Fanuc TP program (LS listing): FM204014.ls

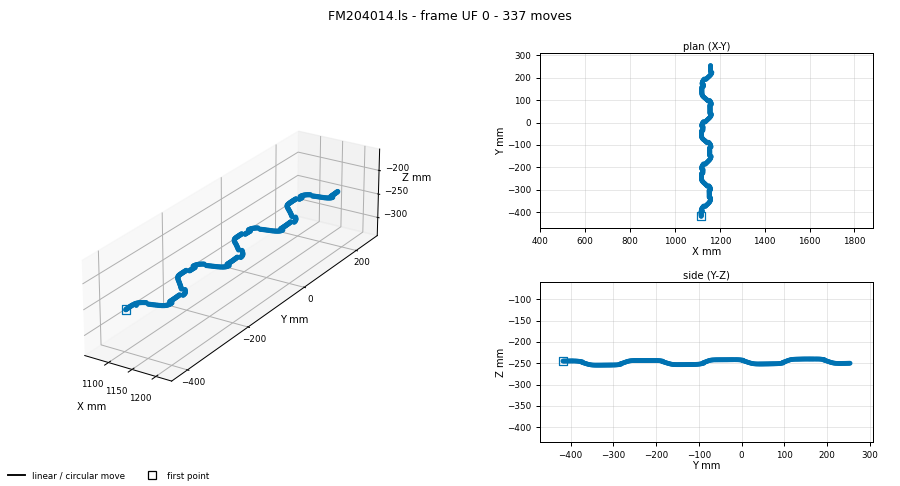
[picture p0: tool path of FM204014.ls in frame UF 0, 337 of 337 moves have a stored position in this frame; points joined in program order, loops and branches not executed]
/PROG  FM204014
/ATTR
OWNER		= MNEDITOR;
COMMENT		= "Auto FANUC move";
PROG_SIZE	= 0;
CREATE		= DATE 26-04-24  TIME 20:40:14;
MODIFIED	= DATE 26-04-24  TIME 20:40:14;
FILE_NAME	= ;
VERSION		= 0;
LINE_COUNT	= 342;
MEMORY_SIZE	= 0;
PROTECT		= READ_WRITE;
TCD:  STACK_SIZE	= 0,
      TASK_PRIORITY	= 50,
      TIME_SLICE	= 0,
      BUSY_LAMP_OFF	= 0,
      ABORT_REQUEST	= 0,
      PAUSE_REQUEST	= 0;
DEFAULT_GROUP	= 1,*,*,*,*;
CONTROL_CODE	= 00000000 00000000;
/MN
   1:  UFRAME_NUM=0 ;
   2:  UTOOL_NUM=1 ;
   3:  R[93]=10 ;
   4:  L P[1] 7mm/sec FINE ;
   5:  L P[2] 7mm/sec CNT50 ;
   6:  L P[3] 7mm/sec CNT50 ;
   7:  L P[4] 7mm/sec CNT50 ;
   8:  L P[5] 7mm/sec CNT50 ;
   9:  L P[6] 7mm/sec CNT50 ;
  10:  L P[7] 7mm/sec CNT50 ;
  11:  L P[8] 7mm/sec CNT50 ;
  12:  L P[9] 7mm/sec CNT50 ;
  13:  L P[10] 7mm/sec CNT50 ;
  14:  L P[11] 7mm/sec CNT50 ;
  15:  L P[12] 7mm/sec CNT50 ;
  16:  L P[13] 7mm/sec CNT50 ;
  17:  L P[14] 7mm/sec CNT50 ;
  18:  L P[15] 7mm/sec CNT50 ;
  19:  L P[16] 7mm/sec CNT50 ;
  20:  L P[17] 7mm/sec CNT50 ;
  21:  L P[18] 7mm/sec CNT50 ;
  22:  L P[19] 7mm/sec CNT50 ;
  23:  L P[20] 7mm/sec CNT50 ;
  24:  L P[21] 7mm/sec CNT50 ;
  25:  L P[22] 7mm/sec CNT50 ;
  26:  L P[23] 7mm/sec CNT50 ;
  27:  L P[24] 7mm/sec CNT50 ;
  28:  L P[25] 7mm/sec CNT50 ;
  29:  L P[26] 7mm/sec CNT50 ;
  30:  L P[27] 7mm/sec CNT50 ;
  31:  L P[28] 7mm/sec CNT50 ;
  32:  L P[29] 7mm/sec CNT50 ;
  33:  L P[30] 7mm/sec CNT50 ;
  34:  L P[31] 7mm/sec CNT50 ;
  35:  L P[32] 7mm/sec CNT50 ;
  36:  L P[33] 7mm/sec CNT50 ;
  37:  L P[34] 7mm/sec CNT50 ;
  38:  L P[35] 7mm/sec CNT50 ;
  39:  L P[36] 7mm/sec CNT50 ;
  40:  L P[37] 7mm/sec CNT50 ;
  41:  L P[38] 7mm/sec CNT50 ;
  42:  L P[39] 7mm/sec CNT50 ;
  43:  L P[40] 7mm/sec CNT50 ;
  44:  L P[41] 7mm/sec CNT50 ;
  45:  L P[42] 7mm/sec CNT50 ;
  46:  L P[43] 7mm/sec CNT50 ;
  47:  L P[44] 7mm/sec CNT50 ;
  48:  L P[45] 7mm/sec CNT50 ;
  49:  L P[46] 7mm/sec CNT50 ;
  50:  L P[47] 7mm/sec CNT50 ;
  51:  L P[48] 7mm/sec CNT50 ;
  52:  L P[49] 7mm/sec CNT50 ;
  53:  L P[50] 7mm/sec CNT50 ;
  54:  L P[51] 7mm/sec CNT50 ;
  55:  L P[52] 7mm/sec CNT50 ;
  56:  L P[53] 7mm/sec CNT50 ;
  57:  L P[54] 7mm/sec CNT50 ;
  58:  L P[55] 7mm/sec CNT50 ;
  59:  L P[56] 7mm/sec CNT50 ;
  60:  L P[57] 7mm/sec CNT50 ;
  61:  L P[58] 7mm/sec CNT50 ;
  62:  L P[59] 7mm/sec CNT50 ;
  63:  L P[60] 7mm/sec CNT50 ;
  64:  L P[61] 7mm/sec CNT50 ;
  65:  L P[62] 7mm/sec CNT50 ;
  66:  L P[63] 7mm/sec CNT50 ;
  67:  L P[64] 7mm/sec CNT50 ;
  68:  L P[65] 7mm/sec CNT50 ;
  69:  L P[66] 7mm/sec CNT50 ;
  70:  L P[67] 7mm/sec CNT50 ;
  71:  L P[68] 7mm/sec CNT50 ;
  72:  L P[69] 7mm/sec CNT50 ;
  73:  L P[70] 7mm/sec CNT50 ;
  74:  L P[71] 7mm/sec CNT50 ;
  75:  L P[72] 7mm/sec CNT50 ;
  76:  L P[73] 7mm/sec CNT50 ;
  77:  L P[74] 7mm/sec CNT50 ;
  78:  L P[75] 7mm/sec CNT50 ;
  79:  L P[76] 7mm/sec CNT50 ;
  80:  L P[77] 7mm/sec CNT50 ;
  81:  L P[78] 7mm/sec CNT50 ;
  82:  L P[79] 7mm/sec CNT50 ;
  83:  L P[80] 7mm/sec CNT50 ;
  84:  L P[81] 7mm/sec CNT50 ;
  85:  L P[82] 7mm/sec CNT50 ;
  86:  L P[83] 7mm/sec CNT50 ;
  87:  L P[84] 7mm/sec CNT50 ;
  88:  L P[85] 7mm/sec CNT50 ;
  89:  L P[86] 7mm/sec CNT50 ;
  90:  L P[87] 7mm/sec CNT50 ;
  91:  L P[88] 7mm/sec CNT50 ;
  92:  L P[89] 7mm/sec CNT50 ;
  93:  L P[90] 7mm/sec CNT50 ;
  94:  L P[91] 7mm/sec CNT50 ;
  95:  L P[92] 7mm/sec CNT50 ;
  96:  L P[93] 7mm/sec CNT50 ;
  97:  L P[94] 7mm/sec CNT50 ;
  98:  L P[95] 7mm/sec CNT50 ;
  99:  L P[96] 7mm/sec CNT50 ;
 100:  L P[97] 7mm/sec CNT50 ;
 101:  L P[98] 7mm/sec CNT50 ;
 102:  L P[99] 7mm/sec CNT50 ;
 103:  L P[100] 7mm/sec CNT50 ;
 104:  L P[101] 7mm/sec CNT50 ;
 105:  L P[102] 7mm/sec CNT50 ;
 106:  L P[103] 7mm/sec CNT50 ;
 107:  L P[104] 7mm/sec CNT50 ;
 108:  L P[105] 7mm/sec CNT50 ;
 109:  L P[106] 7mm/sec CNT50 ;
 110:  L P[107] 7mm/sec CNT50 ;
 111:  L P[108] 7mm/sec CNT50 ;
 112:  L P[109] 7mm/sec CNT50 ;
 113:  L P[110] 7mm/sec CNT50 ;
 114:  L P[111] 7mm/sec CNT50 ;
 115:  L P[112] 7mm/sec CNT50 ;
 116:  L P[113] 7mm/sec CNT50 ;
 117:  L P[114] 7mm/sec CNT50 ;
 118:  L P[115] 7mm/sec CNT50 ;
 119:  L P[116] 7mm/sec CNT50 ;
 120:  L P[117] 7mm/sec CNT50 ;
 121:  L P[118] 7mm/sec CNT50 ;
 122:  L P[119] 7mm/sec CNT50 ;
 123:  L P[120] 7mm/sec CNT50 ;
 124:  L P[121] 7mm/sec CNT50 ;
 125:  L P[122] 7mm/sec CNT50 ;
 126:  L P[123] 7mm/sec CNT50 ;
 127:  L P[124] 7mm/sec CNT50 ;
 128:  L P[125] 7mm/sec CNT50 ;
 129:  L P[126] 7mm/sec CNT50 ;
 130:  L P[127] 7mm/sec CNT50 ;
 131:  L P[128] 7mm/sec CNT50 ;
 132:  L P[129] 7mm/sec CNT50 ;
 133:  L P[130] 7mm/sec CNT50 ;
 134:  L P[131] 7mm/sec CNT50 ;
 135:  L P[132] 7mm/sec CNT50 ;
 136:  L P[133] 7mm/sec CNT50 ;
 137:  L P[134] 7mm/sec CNT50 ;
 138:  L P[135] 7mm/sec CNT50 ;
 139:  L P[136] 7mm/sec CNT50 ;
 140:  L P[137] 7mm/sec CNT50 ;
 141:  L P[138] 7mm/sec CNT50 ;
 142:  L P[139] 7mm/sec CNT50 ;
 143:  L P[140] 7mm/sec CNT50 ;
 144:  L P[141] 7mm/sec CNT50 ;
 145:  L P[142] 7mm/sec CNT50 ;
 146:  L P[143] 7mm/sec CNT50 ;
 147:  L P[144] 7mm/sec CNT50 ;
 148:  L P[145] 7mm/sec CNT50 ;
 149:  L P[146] 7mm/sec CNT50 ;
 150:  L P[147] 7mm/sec CNT50 ;
 151:  L P[148] 7mm/sec CNT50 ;
 152:  L P[149] 7mm/sec CNT50 ;
 153:  L P[150] 7mm/sec CNT50 ;
 154:  L P[151] 7mm/sec CNT50 ;
 155:  L P[152] 7mm/sec CNT50 ;
 156:  L P[153] 7mm/sec CNT50 ;
 157:  L P[154] 7mm/sec CNT50 ;
 158:  L P[155] 7mm/sec CNT50 ;
 159:  L P[156] 7mm/sec CNT50 ;
 160:  L P[157] 7mm/sec CNT50 ;
 161:  L P[158] 7mm/sec CNT50 ;
 162:  L P[159] 7mm/sec CNT50 ;
 163:  L P[160] 7mm/sec CNT50 ;
 164:  L P[161] 7mm/sec CNT50 ;
 165:  L P[162] 7mm/sec CNT50 ;
 166:  L P[163] 7mm/sec CNT50 ;
 167:  L P[164] 7mm/sec CNT50 ;
 168:  L P[165] 7mm/sec CNT50 ;
 169:  L P[166] 7mm/sec CNT50 ;
 170:  L P[167] 7mm/sec CNT50 ;
 171:  L P[168] 7mm/sec CNT50 ;
 172:  L P[169] 7mm/sec CNT50 ;
 173:  L P[170] 7mm/sec CNT50 ;
 174:  L P[171] 7mm/sec CNT50 ;
 175:  L P[172] 7mm/sec CNT50 ;
 176:  L P[173] 7mm/sec CNT50 ;
 177:  L P[174] 7mm/sec CNT50 ;
 178:  L P[175] 7mm/sec CNT50 ;
 179:  L P[176] 7mm/sec CNT50 ;
 180:  L P[177] 7mm/sec CNT50 ;
 181:  L P[178] 7mm/sec CNT50 ;
 182:  L P[179] 7mm/sec CNT50 ;
 183:  L P[180] 7mm/sec CNT50 ;
 184:  L P[181] 7mm/sec CNT50 ;
 185:  L P[182] 7mm/sec CNT50 ;
 186:  L P[183] 7mm/sec CNT50 ;
 187:  L P[184] 7mm/sec CNT50 ;
 188:  L P[185] 7mm/sec CNT50 ;
 189:  L P[186] 7mm/sec CNT50 ;
 190:  L P[187] 7mm/sec CNT50 ;
 191:  L P[188] 7mm/sec CNT50 ;
 192:  L P[189] 7mm/sec CNT50 ;
 193:  L P[190] 7mm/sec CNT50 ;
 194:  L P[191] 7mm/sec CNT50 ;
 195:  L P[192] 7mm/sec CNT50 ;
 196:  L P[193] 7mm/sec CNT50 ;
 197:  L P[194] 7mm/sec CNT50 ;
 198:  L P[195] 7mm/sec CNT50 ;
 199:  L P[196] 7mm/sec CNT50 ;
 200:  L P[197] 7mm/sec CNT50 ;
 201:  L P[198] 7mm/sec CNT50 ;
 202:  L P[199] 7mm/sec CNT50 ;
 203:  L P[200] 7mm/sec CNT50 ;
 204:  L P[201] 7mm/sec CNT50 ;
 205:  L P[202] 7mm/sec CNT50 ;
 206:  L P[203] 7mm/sec CNT50 ;
 207:  L P[204] 7mm/sec CNT50 ;
 208:  L P[205] 7mm/sec CNT50 ;
 209:  L P[206] 7mm/sec CNT50 ;
 210:  L P[207] 7mm/sec CNT50 ;
 211:  L P[208] 7mm/sec CNT50 ;
 212:  L P[209] 7mm/sec CNT50 ;
 213:  L P[210] 7mm/sec CNT50 ;
 214:  L P[211] 7mm/sec CNT50 ;
 215:  L P[212] 7mm/sec CNT50 ;
 216:  L P[213] 7mm/sec CNT50 ;
 217:  L P[214] 7mm/sec CNT50 ;
 218:  L P[215] 7mm/sec CNT50 ;
 219:  L P[216] 7mm/sec CNT50 ;
 220:  L P[217] 7mm/sec CNT50 ;
 221:  L P[218] 7mm/sec CNT50 ;
 222:  L P[219] 7mm/sec CNT50 ;
 223:  L P[220] 7mm/sec CNT50 ;
 224:  L P[221] 7mm/sec CNT50 ;
 225:  L P[222] 7mm/sec CNT50 ;
 226:  L P[223] 7mm/sec CNT50 ;
 227:  L P[224] 7mm/sec CNT50 ;
 228:  L P[225] 7mm/sec CNT50 ;
 229:  L P[226] 7mm/sec CNT50 ;
 230:  L P[227] 7mm/sec CNT50 ;
 231:  L P[228] 7mm/sec CNT50 ;
 232:  L P[229] 7mm/sec CNT50 ;
 233:  L P[230] 7mm/sec CNT50 ;
 234:  L P[231] 7mm/sec CNT50 ;
 235:  L P[232] 7mm/sec CNT50 ;
 236:  L P[233] 7mm/sec CNT50 ;
 237:  L P[234] 7mm/sec CNT50 ;
 238:  L P[235] 7mm/sec CNT50 ;
 239:  L P[236] 7mm/sec CNT50 ;
 240:  L P[237] 7mm/sec CNT50 ;
 241:  L P[238] 7mm/sec CNT50 ;
 242:  L P[239] 7mm/sec CNT50 ;
 243:  L P[240] 7mm/sec CNT50 ;
 244:  L P[241] 7mm/sec CNT50 ;
 245:  L P[242] 7mm/sec CNT50 ;
 246:  L P[243] 7mm/sec CNT50 ;
 247:  L P[244] 7mm/sec CNT50 ;
 248:  L P[245] 7mm/sec CNT50 ;
 249:  L P[246] 7mm/sec CNT50 ;
 250:  L P[247] 7mm/sec CNT50 ;
 251:  L P[248] 7mm/sec CNT50 ;
 252:  L P[249] 7mm/sec CNT50 ;
 253:  L P[250] 7mm/sec CNT50 ;
 254:  L P[251] 7mm/sec CNT50 ;
 255:  L P[252] 7mm/sec CNT50 ;
 256:  L P[253] 7mm/sec CNT50 ;
 257:  L P[254] 7mm/sec CNT50 ;
 258:  L P[255] 7mm/sec CNT50 ;
 259:  L P[256] 7mm/sec CNT50 ;
 260:  L P[257] 7mm/sec CNT50 ;
 261:  L P[258] 7mm/sec CNT50 ;
 262:  L P[259] 7mm/sec CNT50 ;
 263:  L P[260] 7mm/sec CNT50 ;
 264:  L P[261] 7mm/sec CNT50 ;
 265:  L P[262] 7mm/sec CNT50 ;
 266:  L P[263] 7mm/sec CNT50 ;
 267:  L P[264] 7mm/sec CNT50 ;
 268:  L P[265] 7mm/sec CNT50 ;
 269:  L P[266] 7mm/sec CNT50 ;
 270:  L P[267] 7mm/sec CNT50 ;
 271:  L P[268] 7mm/sec CNT50 ;
 272:  L P[269] 7mm/sec CNT50 ;
 273:  L P[270] 7mm/sec CNT50 ;
 274:  L P[271] 7mm/sec CNT50 ;
 275:  L P[272] 7mm/sec CNT50 ;
 276:  L P[273] 7mm/sec CNT50 ;
 277:  L P[274] 7mm/sec CNT50 ;
 278:  L P[275] 7mm/sec CNT50 ;
 279:  L P[276] 7mm/sec CNT50 ;
 280:  L P[277] 7mm/sec CNT50 ;
 281:  L P[278] 7mm/sec CNT50 ;
 282:  L P[279] 7mm/sec CNT50 ;
 283:  L P[280] 7mm/sec CNT50 ;
 284:  L P[281] 7mm/sec CNT50 ;
 285:  L P[282] 7mm/sec CNT50 ;
 286:  L P[283] 7mm/sec CNT50 ;
 287:  L P[284] 7mm/sec CNT50 ;
 288:  L P[285] 7mm/sec CNT50 ;
 289:  L P[286] 7mm/sec CNT50 ;
 290:  L P[287] 7mm/sec CNT50 ;
 291:  L P[288] 7mm/sec CNT50 ;
 292:  L P[289] 7mm/sec CNT50 ;
 293:  L P[290] 7mm/sec CNT50 ;
 294:  L P[291] 7mm/sec CNT50 ;
 295:  L P[292] 7mm/sec CNT50 ;
 296:  L P[293] 7mm/sec CNT50 ;
 297:  L P[294] 7mm/sec CNT50 ;
 298:  L P[295] 7mm/sec CNT50 ;
 299:  L P[296] 7mm/sec CNT50 ;
 300:  L P[297] 7mm/sec CNT50 ;
 301:  L P[298] 7mm/sec CNT50 ;
 302:  L P[299] 7mm/sec CNT50 ;
 303:  L P[300] 7mm/sec CNT50 ;
 304:  L P[301] 7mm/sec CNT50 ;
 305:  L P[302] 7mm/sec CNT50 ;
 306:  L P[303] 7mm/sec CNT50 ;
 307:  L P[304] 7mm/sec CNT50 ;
 308:  L P[305] 7mm/sec CNT50 ;
 309:  L P[306] 7mm/sec CNT50 ;
 310:  L P[307] 7mm/sec CNT50 ;
 311:  L P[308] 7mm/sec CNT50 ;
 312:  L P[309] 7mm/sec CNT50 ;
 313:  L P[310] 7mm/sec CNT50 ;
 314:  L P[311] 7mm/sec CNT50 ;
 315:  L P[312] 7mm/sec CNT50 ;
 316:  L P[313] 7mm/sec CNT50 ;
 317:  L P[314] 7mm/sec CNT50 ;
 318:  L P[315] 7mm/sec CNT50 ;
 319:  L P[316] 7mm/sec CNT50 ;
 320:  L P[317] 7mm/sec CNT50 ;
 321:  L P[318] 7mm/sec CNT50 ;
 322:  L P[319] 7mm/sec CNT50 ;
 323:  L P[320] 7mm/sec CNT50 ;
 324:  L P[321] 7mm/sec CNT50 ;
 325:  L P[322] 7mm/sec CNT50 ;
 326:  L P[323] 7mm/sec CNT50 ;
 327:  L P[324] 7mm/sec CNT50 ;
 328:  L P[325] 7mm/sec CNT50 ;
 329:  L P[326] 7mm/sec CNT50 ;
 330:  L P[327] 7mm/sec CNT50 ;
 331:  L P[328] 7mm/sec CNT50 ;
 332:  L P[329] 7mm/sec CNT50 ;
 333:  L P[330] 7mm/sec CNT50 ;
 334:  L P[331] 7mm/sec CNT50 ;
 335:  L P[332] 7mm/sec CNT50 ;
 336:  L P[333] 7mm/sec CNT50 ;
 337:  L P[334] 7mm/sec CNT50 ;
 338:  L P[335] 7mm/sec CNT50 ;
 339:  L P[336] 7mm/sec CNT50 ;
 340:  L P[337] 7mm/sec FINE ;
 341:  R[93]=1 ;
 342:  END ;
/POS
P[1]{
   GP1:
	UF : 0, UT : 1,		CONFIG : 'N U T, 0, 0, 0',
	X = 1117.340  mm,	Y = -418.120  mm,	Z = -244.843  mm,
	W = 0.000 deg,	P = 30.000 deg,	R = 175.540 deg
};
P[2]{
   GP1:
	UF : 0, UT : 1,		CONFIG : 'N U T, 0, 0, 0',
	X = 1117.260  mm,	Y = -416.121  mm,	Z = -244.824  mm,
	W = 0.000 deg,	P = 30.000 deg,	R = 175.540 deg
};
P[3]{
   GP1:
	UF : 0, UT : 1,		CONFIG : 'N U T, 0, 0, 0',
	X = 1117.178  mm,	Y = -414.124  mm,	Z = -244.789  mm,
	W = 0.000 deg,	P = 30.000 deg,	R = 175.540 deg
};
P[4]{
   GP1:
	UF : 0, UT : 1,		CONFIG : 'N U T, 0, 0, 0',
	X = 1117.094  mm,	Y = -412.119  mm,	Z = -244.747  mm,
	W = 0.000 deg,	P = 30.000 deg,	R = 175.540 deg
};
P[5]{
   GP1:
	UF : 0, UT : 1,		CONFIG : 'N U T, 0, 0, 0',
	X = 1117.019  mm,	Y = -410.103  mm,	Z = -244.710  mm,
	W = 0.000 deg,	P = 30.000 deg,	R = 175.540 deg
};
P[6]{
   GP1:
	UF : 0, UT : 1,		CONFIG : 'N U T, 0, 0, 0',
	X = 1116.955  mm,	Y = -408.082  mm,	Z = -244.672  mm,
	W = 0.000 deg,	P = 30.000 deg,	R = 175.540 deg
};
P[7]{
   GP1:
	UF : 0, UT : 1,		CONFIG : 'N U T, 0, 0, 0',
	X = 1116.909  mm,	Y = -406.055  mm,	Z = -244.633  mm,
	W = 0.000 deg,	P = 30.000 deg,	R = 175.540 deg
};
P[8]{
   GP1:
	UF : 0, UT : 1,		CONFIG : 'N U T, 0, 0, 0',
	X = 1116.881  mm,	Y = -404.021  mm,	Z = -244.596  mm,
	W = 0.000 deg,	P = 30.000 deg,	R = 175.540 deg
};
P[9]{
   GP1:
	UF : 0, UT : 1,		CONFIG : 'N U T, 0, 0, 0',
	X = 1116.880  mm,	Y = -401.987  mm,	Z = -244.564  mm,
	W = 0.000 deg,	P = 30.000 deg,	R = 175.540 deg
};
P[10]{
   GP1:
	UF : 0, UT : 1,		CONFIG : 'N U T, 0, 0, 0',
	X = 1116.899  mm,	Y = -399.955  mm,	Z = -244.547  mm,
	W = 0.000 deg,	P = 30.000 deg,	R = 175.540 deg
};
P[11]{
   GP1:
	UF : 0, UT : 1,		CONFIG : 'N U T, 0, 0, 0',
	X = 1116.941  mm,	Y = -397.902  mm,	Z = -244.542  mm,
	W = 0.000 deg,	P = 30.000 deg,	R = 175.540 deg
};
P[12]{
   GP1:
	UF : 0, UT : 1,		CONFIG : 'N U T, 0, 0, 0',
	X = 1117.034  mm,	Y = -395.846  mm,	Z = -244.547  mm,
	W = 0.000 deg,	P = 30.000 deg,	R = 175.540 deg
};
P[13]{
   GP1:
	UF : 0, UT : 1,		CONFIG : 'N U T, 0, 0, 0',
	X = 1123.135  mm,	Y = -394.244  mm,	Z = -244.557  mm,
	W = 0.000 deg,	P = 30.000 deg,	R = 175.540 deg
};
P[14]{
   GP1:
	UF : 0, UT : 1,		CONFIG : 'N U T, 0, 0, 0',
	X = 1117.391  mm,	Y = -391.546  mm,	Z = -244.600  mm,
	W = 0.000 deg,	P = 30.000 deg,	R = 169.940 deg
};
P[15]{
   GP1:
	UF : 0, UT : 1,		CONFIG : 'N U T, 0, 0, 0',
	X = 1117.843  mm,	Y = -389.291  mm,	Z = -244.691  mm,
	W = 0.000 deg,	P = 30.000 deg,	R = 162.053 deg
};
P[16]{
   GP1:
	UF : 0, UT : 1,		CONFIG : 'N U T, 0, 0, 0',
	X = 1118.496  mm,	Y = -387.015  mm,	Z = -244.808  mm,
	W = 0.000 deg,	P = 30.000 deg,	R = 154.006 deg
};
P[17]{
   GP1:
	UF : 0, UT : 1,		CONFIG : 'N U T, 0, 0, 0',
	X = 1119.426  mm,	Y = -384.740  mm,	Z = -244.961  mm,
	W = 0.000 deg,	P = 30.000 deg,	R = 145.637 deg
};
P[18]{
   GP1:
	UF : 0, UT : 1,		CONFIG : 'N U T, 0, 0, 0',
	X = 1120.551  mm,	Y = -382.554  mm,	Z = -245.152  mm,
	W = 0.000 deg,	P = 30.000 deg,	R = 136.915 deg
};
P[19]{
   GP1:
	UF : 0, UT : 1,		CONFIG : 'N U T, 0, 0, 0',
	X = 1121.835  mm,	Y = -380.363  mm,	Z = -245.385  mm,
	W = 0.000 deg,	P = 30.000 deg,	R = 136.915 deg
};
P[20]{
   GP1:
	UF : 0, UT : 1,		CONFIG : 'N U T, 0, 0, 0',
	X = 1123.398  mm,	Y = -378.182  mm,	Z = -245.708  mm,
	W = 0.000 deg,	P = 30.000 deg,	R = 136.915 deg
};
P[21]{
   GP1:
	UF : 0, UT : 1,		CONFIG : 'N U T, 0, 0, 0',
	X = 1125.083  mm,	Y = -376.092  mm,	Z = -246.105  mm,
	W = 0.000 deg,	P = 30.000 deg,	R = 136.915 deg
};
P[22]{
   GP1:
	UF : 0, UT : 1,		CONFIG : 'N U T, 0, 0, 0',
	X = 1126.825  mm,	Y = -374.022  mm,	Z = -246.540  mm,
	W = 0.000 deg,	P = 30.000 deg,	R = 136.915 deg
};
P[23]{
   GP1:
	UF : 0, UT : 1,		CONFIG : 'N U T, 0, 0, 0',
	X = 1128.702  mm,	Y = -371.963  mm,	Z = -247.047  mm,
	W = 0.000 deg,	P = 30.000 deg,	R = 136.915 deg
};
P[24]{
   GP1:
	UF : 0, UT : 1,		CONFIG : 'N U T, 0, 0, 0',
	X = 1134.942  mm,	Y = -374.080  mm,	Z = -247.615  mm,
	W = 0.000 deg,	P = 30.000 deg,	R = 136.915 deg
};
P[25]{
   GP1:
	UF : 0, UT : 1,		CONFIG : 'N U T, 0, 0, 0',
	X = 1136.860  mm,	Y = -372.134  mm,	Z = -248.238  mm,
	W = 0.000 deg,	P = 30.000 deg,	R = 136.915 deg
};
P[26]{
   GP1:
	UF : 0, UT : 1,		CONFIG : 'N U T, 0, 0, 0',
	X = 1138.910  mm,	Y = -370.162  mm,	Z = -248.902  mm,
	W = 0.000 deg,	P = 30.000 deg,	R = 136.915 deg
};
P[27]{
   GP1:
	UF : 0, UT : 1,		CONFIG : 'N U T, 0, 0, 0',
	X = 1140.982  mm,	Y = -368.168  mm,	Z = -249.556  mm,
	W = 0.000 deg,	P = 30.000 deg,	R = 136.915 deg
};
P[28]{
   GP1:
	UF : 0, UT : 1,		CONFIG : 'N U T, 0, 0, 0',
	X = 1143.070  mm,	Y = -366.183  mm,	Z = -250.199  mm,
	W = 0.000 deg,	P = 30.000 deg,	R = 136.915 deg
};
P[29]{
   GP1:
	UF : 0, UT : 1,		CONFIG : 'N U T, 0, 0, 0',
	X = 1145.207  mm,	Y = -364.186  mm,	Z = -250.847  mm,
	W = 0.000 deg,	P = 30.000 deg,	R = 136.915 deg
};
P[30]{
   GP1:
	UF : 0, UT : 1,		CONFIG : 'N U T, 0, 0, 0',
	X = 1147.334  mm,	Y = -362.176  mm,	Z = -251.475  mm,
	W = 0.000 deg,	P = 30.000 deg,	R = 143.608 deg
};
P[31]{
   GP1:
	UF : 0, UT : 1,		CONFIG : 'N U T, 0, 0, 0',
	X = 1149.502  mm,	Y = -360.107  mm,	Z = -252.087  mm,
	W = 0.000 deg,	P = 30.000 deg,	R = 156.114 deg
};
P[32]{
   GP1:
	UF : 0, UT : 1,		CONFIG : 'N U T, 0, 0, 0',
	X = 1151.458  mm,	Y = -357.994  mm,	Z = -252.623  mm,
	W = 0.000 deg,	P = 30.000 deg,	R = 167.837 deg
};
P[33]{
   GP1:
	UF : 0, UT : 1,		CONFIG : 'N U T, 0, 0, 0',
	X = 1153.272  mm,	Y = -355.871  mm,	Z = -253.109  mm,
	W = 0.000 deg,	P = 30.000 deg,	R = 179.135 deg
};
P[34]{
   GP1:
	UF : 0, UT : 1,		CONFIG : 'N U T, 0, 0, 0',
	X = 1154.901  mm,	Y = -353.669  mm,	Z = -253.519  mm,
	W = 0.000 deg,	P = 30.000 deg,	R = 179.135 deg
};
P[35]{
   GP1:
	UF : 0, UT : 1,		CONFIG : 'N U T, 0, 0, 0',
	X = 1156.258  mm,	Y = -351.400  mm,	Z = -253.841  mm,
	W = 0.000 deg,	P = 30.000 deg,	R = 179.135 deg
};
P[36]{
   GP1:
	UF : 0, UT : 1,		CONFIG : 'N U T, 0, 0, 0',
	X = 1157.318  mm,	Y = -349.081  mm,	Z = -254.072  mm,
	W = 0.000 deg,	P = 30.000 deg,	R = 179.135 deg
};
P[37]{
   GP1:
	UF : 0, UT : 1,		CONFIG : 'N U T, 0, 0, 0',
	X = 1158.065  mm,	Y = -346.706  mm,	Z = -254.224  mm,
	W = 0.000 deg,	P = 30.000 deg,	R = 179.135 deg
};
P[38]{
   GP1:
	UF : 0, UT : 1,		CONFIG : 'N U T, 0, 0, 0',
	X = 1158.455  mm,	Y = -344.449  mm,	Z = -254.296  mm,
	W = 0.000 deg,	P = 30.000 deg,	R = 179.135 deg
};
P[39]{
   GP1:
	UF : 0, UT : 1,		CONFIG : 'N U T, 0, 0, 0',
	X = 1158.742  mm,	Y = -342.283  mm,	Z = -254.346  mm,
	W = 0.000 deg,	P = 30.000 deg,	R = 179.135 deg
};
P[40]{
   GP1:
	UF : 0, UT : 1,		CONFIG : 'N U T, 0, 0, 0',
	X = 1158.865  mm,	Y = -340.124  mm,	Z = -254.355  mm,
	W = 0.000 deg,	P = 30.000 deg,	R = 179.135 deg
};
P[41]{
   GP1:
	UF : 0, UT : 1,		CONFIG : 'N U T, 0, 0, 0',
	X = 1158.920  mm,	Y = -338.068  mm,	Z = -254.355  mm,
	W = 0.000 deg,	P = 30.000 deg,	R = 179.135 deg
};
P[42]{
   GP1:
	UF : 0, UT : 1,		CONFIG : 'N U T, 0, 0, 0',
	X = 1158.958  mm,	Y = -336.046  mm,	Z = -254.353  mm,
	W = 0.000 deg,	P = 30.000 deg,	R = 179.135 deg
};
P[43]{
   GP1:
	UF : 0, UT : 1,		CONFIG : 'N U T, 0, 0, 0',
	X = 1152.982  mm,	Y = -333.969  mm,	Z = -254.350  mm,
	W = 0.000 deg,	P = 30.000 deg,	R = 179.135 deg
};
P[44]{
   GP1:
	UF : 0, UT : 1,		CONFIG : 'N U T, 0, 0, 0',
	X = 1153.000  mm,	Y = -331.976  mm,	Z = -254.343  mm,
	W = 0.000 deg,	P = 30.000 deg,	R = 179.135 deg
};
P[45]{
   GP1:
	UF : 0, UT : 1,		CONFIG : 'N U T, 0, 0, 0',
	X = 1153.014  mm,	Y = -329.984  mm,	Z = -254.328  mm,
	W = 0.000 deg,	P = 30.000 deg,	R = 179.135 deg
};
P[46]{
   GP1:
	UF : 0, UT : 1,		CONFIG : 'N U T, 0, 0, 0',
	X = 1153.021  mm,	Y = -327.991  mm,	Z = -254.312  mm,
	W = 0.000 deg,	P = 30.000 deg,	R = 179.135 deg
};
P[47]{
   GP1:
	UF : 0, UT : 1,		CONFIG : 'N U T, 0, 0, 0',
	X = 1153.026  mm,	Y = -325.995  mm,	Z = -254.292  mm,
	W = 0.000 deg,	P = 30.000 deg,	R = 179.135 deg
};
P[48]{
   GP1:
	UF : 0, UT : 1,		CONFIG : 'N U T, 0, 0, 0',
	X = 1153.029  mm,	Y = -323.998  mm,	Z = -254.272  mm,
	W = 0.000 deg,	P = 30.000 deg,	R = 179.135 deg
};
P[49]{
   GP1:
	UF : 0, UT : 1,		CONFIG : 'N U T, 0, 0, 0',
	X = 1153.029  mm,	Y = -322.001  mm,	Z = -254.251  mm,
	W = 0.000 deg,	P = 30.000 deg,	R = 179.135 deg
};
P[50]{
   GP1:
	UF : 0, UT : 1,		CONFIG : 'N U T, 0, 0, 0',
	X = 1153.027  mm,	Y = -320.008  mm,	Z = -254.230  mm,
	W = 0.000 deg,	P = 30.000 deg,	R = 179.135 deg
};
P[51]{
   GP1:
	UF : 0, UT : 1,		CONFIG : 'N U T, 0, 0, 0',
	X = 1153.018  mm,	Y = -318.016  mm,	Z = -254.210  mm,
	W = 0.000 deg,	P = 30.000 deg,	R = 179.135 deg
};
P[52]{
   GP1:
	UF : 0, UT : 1,		CONFIG : 'N U T, 0, 0, 0',
	X = 1153.005  mm,	Y = -316.026  mm,	Z = -254.197  mm,
	W = 0.000 deg,	P = 30.000 deg,	R = 179.135 deg
};
P[53]{
   GP1:
	UF : 0, UT : 1,		CONFIG : 'N U T, 0, 0, 0',
	X = 1152.983  mm,	Y = -314.037  mm,	Z = -254.183  mm,
	W = 0.000 deg,	P = 30.000 deg,	R = 179.135 deg
};
P[54]{
   GP1:
	UF : 0, UT : 1,		CONFIG : 'N U T, 0, 0, 0',
	X = 1152.956  mm,	Y = -312.053  mm,	Z = -254.171  mm,
	W = 0.000 deg,	P = 30.000 deg,	R = 179.135 deg
};
P[55]{
   GP1:
	UF : 0, UT : 1,		CONFIG : 'N U T, 0, 0, 0',
	X = 1152.913  mm,	Y = -310.069  mm,	Z = -254.154  mm,
	W = 0.000 deg,	P = 30.000 deg,	R = 179.135 deg
};
P[56]{
   GP1:
	UF : 0, UT : 1,		CONFIG : 'N U T, 0, 0, 0',
	X = 1152.865  mm,	Y = -308.079  mm,	Z = -254.132  mm,
	W = 0.000 deg,	P = 30.000 deg,	R = 179.135 deg
};
P[57]{
   GP1:
	UF : 0, UT : 1,		CONFIG : 'N U T, 0, 0, 0',
	X = 1152.808  mm,	Y = -306.093  mm,	Z = -254.108  mm,
	W = 0.000 deg,	P = 30.000 deg,	R = 179.135 deg
};
P[58]{
   GP1:
	UF : 0, UT : 1,		CONFIG : 'N U T, 0, 0, 0',
	X = 1152.742  mm,	Y = -304.113  mm,	Z = -254.081  mm,
	W = 0.000 deg,	P = 30.000 deg,	R = 179.135 deg
};
P[59]{
   GP1:
	UF : 0, UT : 1,		CONFIG : 'N U T, 0, 0, 0',
	X = 1152.659  mm,	Y = -302.131  mm,	Z = -254.050  mm,
	W = 0.000 deg,	P = 30.000 deg,	R = 179.135 deg
};
P[60]{
   GP1:
	UF : 0, UT : 1,		CONFIG : 'N U T, 0, 0, 0',
	X = 1158.558  mm,	Y = -299.816  mm,	Z = -254.014  mm,
	W = 0.000 deg,	P = 30.000 deg,	R = -172.618 deg
};
P[61]{
   GP1:
	UF : 0, UT : 1,		CONFIG : 'N U T, 0, 0, 0',
	X = 1158.403  mm,	Y = -297.780  mm,	Z = -253.956  mm,
	W = 0.000 deg,	P = 30.000 deg,	R = -163.858 deg
};
P[62]{
   GP1:
	UF : 0, UT : 1,		CONFIG : 'N U T, 0, 0, 0',
	X = 1158.252  mm,	Y = -295.667  mm,	Z = -253.904  mm,
	W = 0.000 deg,	P = 30.000 deg,	R = -155.103 deg
};
P[63]{
   GP1:
	UF : 0, UT : 1,		CONFIG : 'N U T, 0, 0, 0',
	X = 1157.902  mm,	Y = -293.394  mm,	Z = -253.806  mm,
	W = 0.000 deg,	P = 30.000 deg,	R = -146.261 deg
};
P[64]{
   GP1:
	UF : 0, UT : 1,		CONFIG : 'N U T, 0, 0, 0',
	X = 1157.226  mm,	Y = -290.874  mm,	Z = -253.644  mm,
	W = 0.000 deg,	P = 30.000 deg,	R = -137.214 deg
};
P[65]{
   GP1:
	UF : 0, UT : 1,		CONFIG : 'N U T, 0, 0, 0',
	X = 1155.922  mm,	Y = -288.464  mm,	Z = -253.306  mm,
	W = 0.000 deg,	P = 30.000 deg,	R = -137.214 deg
};
P[66]{
   GP1:
	UF : 0, UT : 1,		CONFIG : 'N U T, 0, 0, 0',
	X = 1154.539  mm,	Y = -286.310  mm,	Z = -252.913  mm,
	W = 0.000 deg,	P = 30.000 deg,	R = -137.214 deg
};
P[67]{
   GP1:
	UF : 0, UT : 1,		CONFIG : 'N U T, 0, 0, 0',
	X = 1152.984  mm,	Y = -284.157  mm,	Z = -252.468  mm,
	W = 0.000 deg,	P = 30.000 deg,	R = -137.214 deg
};
P[68]{
   GP1:
	UF : 0, UT : 1,		CONFIG : 'N U T, 0, 0, 0',
	X = 1151.189  mm,	Y = -282.007  mm,	Z = -251.954  mm,
	W = 0.000 deg,	P = 30.000 deg,	R = -137.214 deg
};
P[69]{
   GP1:
	UF : 0, UT : 1,		CONFIG : 'N U T, 0, 0, 0',
	X = 1144.873  mm,	Y = -284.051  mm,	Z = -251.372  mm,
	W = 0.000 deg,	P = 30.000 deg,	R = -137.214 deg
};
P[70]{
   GP1:
	UF : 0, UT : 1,		CONFIG : 'N U T, 0, 0, 0',
	X = 1143.084  mm,	Y = -282.127  mm,	Z = -250.789  mm,
	W = 0.000 deg,	P = 30.000 deg,	R = -137.214 deg
};
P[71]{
   GP1:
	UF : 0, UT : 1,		CONFIG : 'N U T, 0, 0, 0',
	X = 1140.897  mm,	Y = -280.100  mm,	Z = -250.108  mm,
	W = 0.000 deg,	P = 30.000 deg,	R = -137.214 deg
};
P[72]{
   GP1:
	UF : 0, UT : 1,		CONFIG : 'N U T, 0, 0, 0',
	X = 1139.113  mm,	Y = -278.077  mm,	Z = -249.543  mm,
	W = 0.000 deg,	P = 30.000 deg,	R = -137.214 deg
};
P[73]{
   GP1:
	UF : 0, UT : 1,		CONFIG : 'N U T, 0, 0, 0',
	X = 1137.130  mm,	Y = -276.172  mm,	Z = -248.855  mm,
	W = 0.000 deg,	P = 30.000 deg,	R = -137.214 deg
};
P[74]{
   GP1:
	UF : 0, UT : 1,		CONFIG : 'N U T, 0, 0, 0',
	X = 1135.018  mm,	Y = -274.181  mm,	Z = -248.131  mm,
	W = 0.000 deg,	P = 30.000 deg,	R = -137.214 deg
};
P[75]{
   GP1:
	UF : 0, UT : 1,		CONFIG : 'N U T, 0, 0, 0',
	X = 1132.885  mm,	Y = -272.164  mm,	Z = -247.407  mm,
	W = 0.000 deg,	P = 30.000 deg,	R = -137.214 deg
};
P[76]{
   GP1:
	UF : 0, UT : 1,		CONFIG : 'N U T, 0, 0, 0',
	X = 1130.904  mm,	Y = -270.230  mm,	Z = -246.722  mm,
	W = 0.000 deg,	P = 30.000 deg,	R = -137.214 deg
};
P[77]{
   GP1:
	UF : 0, UT : 1,		CONFIG : 'N U T, 0, 0, 0',
	X = 1128.507  mm,	Y = -268.227  mm,	Z = -246.003  mm,
	W = 0.000 deg,	P = 30.000 deg,	R = -144.478 deg
};
P[78]{
   GP1:
	UF : 0, UT : 1,		CONFIG : 'N U T, 0, 0, 0',
	X = 1126.363  mm,	Y = -266.129  mm,	Z = -245.406  mm,
	W = 0.000 deg,	P = 30.000 deg,	R = -157.037 deg
};
P[79]{
   GP1:
	UF : 0, UT : 1,		CONFIG : 'N U T, 0, 0, 0',
	X = 1124.222  mm,	Y = -263.965  mm,	Z = -244.835  mm,
	W = 0.000 deg,	P = 30.000 deg,	R = -169.422 deg
};
P[80]{
   GP1:
	UF : 0, UT : 1,		CONFIG : 'N U T, 0, 0, 0',
	X = 1122.542  mm,	Y = -261.705  mm,	Z = -244.449  mm,
	W = 0.000 deg,	P = 30.000 deg,	R = 179.744 deg
};
P[81]{
   GP1:
	UF : 0, UT : 1,		CONFIG : 'N U T, 0, 0, 0',
	X = 1121.122  mm,	Y = -259.488  mm,	Z = -244.141  mm,
	W = 0.000 deg,	P = 30.000 deg,	R = 179.744 deg
};
P[82]{
   GP1:
	UF : 0, UT : 1,		CONFIG : 'N U T, 0, 0, 0',
	X = 1120.002  mm,	Y = -257.260  mm,	Z = -243.919  mm,
	W = 0.000 deg,	P = 30.000 deg,	R = 179.744 deg
};
P[83]{
   GP1:
	UF : 0, UT : 1,		CONFIG : 'N U T, 0, 0, 0',
	X = 1119.004  mm,	Y = -254.866  mm,	Z = -243.728  mm,
	W = 0.000 deg,	P = 30.000 deg,	R = 179.744 deg
};
P[84]{
   GP1:
	UF : 0, UT : 1,		CONFIG : 'N U T, 0, 0, 0',
	X = 1118.547  mm,	Y = -252.407  mm,	Z = -243.620  mm,
	W = 0.000 deg,	P = 30.000 deg,	R = 179.744 deg
};
P[85]{
   GP1:
	UF : 0, UT : 1,		CONFIG : 'N U T, 0, 0, 0',
	X = 1118.334  mm,	Y = -250.175  mm,	Z = -243.548  mm,
	W = 0.000 deg,	P = 30.000 deg,	R = 179.744 deg
};
P[86]{
   GP1:
	UF : 0, UT : 1,		CONFIG : 'N U T, 0, 0, 0',
	X = 1118.285  mm,	Y = -248.059  mm,	Z = -243.512  mm,
	W = 0.000 deg,	P = 30.000 deg,	R = 179.744 deg
};
P[87]{
   GP1:
	UF : 0, UT : 1,		CONFIG : 'N U T, 0, 0, 0',
	X = 1118.250  mm,	Y = -246.031  mm,	Z = -243.474  mm,
	W = 0.000 deg,	P = 30.000 deg,	R = 179.744 deg
};
P[88]{
   GP1:
	UF : 0, UT : 1,		CONFIG : 'N U T, 0, 0, 0',
	X = 1118.244  mm,	Y = -244.004  mm,	Z = -243.451  mm,
	W = 0.000 deg,	P = 30.000 deg,	R = 179.744 deg
};
P[89]{
   GP1:
	UF : 0, UT : 1,		CONFIG : 'N U T, 0, 0, 0',
	X = 1118.244  mm,	Y = -241.998  mm,	Z = -243.432  mm,
	W = 0.000 deg,	P = 30.000 deg,	R = 179.744 deg
};
P[90]{
   GP1:
	UF : 0, UT : 1,		CONFIG : 'N U T, 0, 0, 0',
	X = 1118.246  mm,	Y = -239.997  mm,	Z = -243.414  mm,
	W = 0.000 deg,	P = 30.000 deg,	R = 179.744 deg
};
P[91]{
   GP1:
	UF : 0, UT : 1,		CONFIG : 'N U T, 0, 0, 0',
	X = 1118.248  mm,	Y = -237.996  mm,	Z = -243.394  mm,
	W = 0.000 deg,	P = 30.000 deg,	R = 179.744 deg
};
P[92]{
   GP1:
	UF : 0, UT : 1,		CONFIG : 'N U T, 0, 0, 0',
	X = 1118.252  mm,	Y = -235.995  mm,	Z = -243.381  mm,
	W = 0.000 deg,	P = 30.000 deg,	R = 179.744 deg
};
P[93]{
   GP1:
	UF : 0, UT : 1,		CONFIG : 'N U T, 0, 0, 0',
	X = 1118.255  mm,	Y = -233.994  mm,	Z = -243.374  mm,
	W = 0.000 deg,	P = 30.000 deg,	R = 179.744 deg
};
P[94]{
   GP1:
	UF : 0, UT : 1,		CONFIG : 'N U T, 0, 0, 0',
	X = 1118.260  mm,	Y = -231.993  mm,	Z = -243.366  mm,
	W = 0.000 deg,	P = 30.000 deg,	R = 179.744 deg
};
P[95]{
   GP1:
	UF : 0, UT : 1,		CONFIG : 'N U T, 0, 0, 0',
	X = 1118.265  mm,	Y = -229.993  mm,	Z = -243.358  mm,
	W = 0.000 deg,	P = 30.000 deg,	R = 179.744 deg
};
P[96]{
   GP1:
	UF : 0, UT : 1,		CONFIG : 'N U T, 0, 0, 0',
	X = 1118.269  mm,	Y = -227.990  mm,	Z = -243.350  mm,
	W = 0.000 deg,	P = 30.000 deg,	R = 179.744 deg
};
P[97]{
   GP1:
	UF : 0, UT : 1,		CONFIG : 'N U T, 0, 0, 0',
	X = 1124.278  mm,	Y = -226.021  mm,	Z = -243.343  mm,
	W = 0.000 deg,	P = 30.000 deg,	R = 179.744 deg
};
P[98]{
   GP1:
	UF : 0, UT : 1,		CONFIG : 'N U T, 0, 0, 0',
	X = 1124.297  mm,	Y = -224.035  mm,	Z = -243.335  mm,
	W = 0.000 deg,	P = 30.000 deg,	R = 179.744 deg
};
P[99]{
   GP1:
	UF : 0, UT : 1,		CONFIG : 'N U T, 0, 0, 0',
	X = 1124.325  mm,	Y = -222.045  mm,	Z = -243.326  mm,
	W = 0.000 deg,	P = 30.000 deg,	R = 179.744 deg
};
P[100]{
   GP1:
	UF : 0, UT : 1,		CONFIG : 'N U T, 0, 0, 0',
	X = 1124.357  mm,	Y = -220.054  mm,	Z = -243.314  mm,
	W = 0.000 deg,	P = 30.000 deg,	R = 179.744 deg
};
P[101]{
   GP1:
	UF : 0, UT : 1,		CONFIG : 'N U T, 0, 0, 0',
	X = 1124.397  mm,	Y = -218.069  mm,	Z = -243.304  mm,
	W = 0.000 deg,	P = 30.000 deg,	R = 179.744 deg
};
P[102]{
   GP1:
	UF : 0, UT : 1,		CONFIG : 'N U T, 0, 0, 0',
	X = 1124.449  mm,	Y = -216.086  mm,	Z = -243.293  mm,
	W = 0.000 deg,	P = 30.000 deg,	R = 179.744 deg
};
P[103]{
   GP1:
	UF : 0, UT : 1,		CONFIG : 'N U T, 0, 0, 0',
	X = 1124.511  mm,	Y = -214.103  mm,	Z = -243.286  mm,
	W = 0.000 deg,	P = 30.000 deg,	R = 179.744 deg
};
P[104]{
   GP1:
	UF : 0, UT : 1,		CONFIG : 'N U T, 0, 0, 0',
	X = 1124.586  mm,	Y = -212.117  mm,	Z = -243.282  mm,
	W = 0.000 deg,	P = 30.000 deg,	R = 179.744 deg
};
P[105]{
   GP1:
	UF : 0, UT : 1,		CONFIG : 'N U T, 0, 0, 0',
	X = 1124.666  mm,	Y = -210.135  mm,	Z = -243.281  mm,
	W = 0.000 deg,	P = 30.000 deg,	R = 179.744 deg
};
P[106]{
   GP1:
	UF : 0, UT : 1,		CONFIG : 'N U T, 0, 0, 0',
	X = 1124.763  mm,	Y = -208.176  mm,	Z = -243.288  mm,
	W = 0.000 deg,	P = 30.000 deg,	R = 179.744 deg
};
P[107]{
   GP1:
	UF : 0, UT : 1,		CONFIG : 'N U T, 0, 0, 0',
	X = 1118.914  mm,	Y = -205.764  mm,	Z = -243.301  mm,
	W = 0.000 deg,	P = 30.000 deg,	R = 172.062 deg
};
P[108]{
   GP1:
	UF : 0, UT : 1,		CONFIG : 'N U T, 0, 0, 0',
	X = 1119.100  mm,	Y = -203.691  mm,	Z = -243.322  mm,
	W = 0.000 deg,	P = 30.000 deg,	R = 163.764 deg
};
P[109]{
   GP1:
	UF : 0, UT : 1,		CONFIG : 'N U T, 0, 0, 0',
	X = 1119.351  mm,	Y = -201.564  mm,	Z = -243.362  mm,
	W = 0.000 deg,	P = 30.000 deg,	R = 155.441 deg
};
P[110]{
   GP1:
	UF : 0, UT : 1,		CONFIG : 'N U T, 0, 0, 0',
	X = 1119.750  mm,	Y = -199.318  mm,	Z = -243.436  mm,
	W = 0.000 deg,	P = 30.000 deg,	R = 147.044 deg
};
P[111]{
   GP1:
	UF : 0, UT : 1,		CONFIG : 'N U T, 0, 0, 0',
	X = 1120.406  mm,	Y = -197.052  mm,	Z = -243.564  mm,
	W = 0.000 deg,	P = 30.000 deg,	R = 138.421 deg
};
P[112]{
   GP1:
	UF : 0, UT : 1,		CONFIG : 'N U T, 0, 0, 0',
	X = 1121.239  mm,	Y = -194.836  mm,	Z = -243.726  mm,
	W = 0.000 deg,	P = 30.000 deg,	R = 138.421 deg
};
P[113]{
   GP1:
	UF : 0, UT : 1,		CONFIG : 'N U T, 0, 0, 0',
	X = 1122.274  mm,	Y = -192.617  mm,	Z = -243.904  mm,
	W = 0.000 deg,	P = 30.000 deg,	R = 138.421 deg
};
P[114]{
   GP1:
	UF : 0, UT : 1,		CONFIG : 'N U T, 0, 0, 0',
	X = 1123.542  mm,	Y = -190.405  mm,	Z = -244.135  mm,
	W = 0.000 deg,	P = 30.000 deg,	R = 138.421 deg
};
P[115]{
   GP1:
	UF : 0, UT : 1,		CONFIG : 'N U T, 0, 0, 0',
	X = 1125.012  mm,	Y = -188.246  mm,	Z = -244.455  mm,
	W = 0.000 deg,	P = 30.000 deg,	R = 138.421 deg
};
P[116]{
   GP1:
	UF : 0, UT : 1,		CONFIG : 'N U T, 0, 0, 0',
	X = 1126.637  mm,	Y = -186.110  mm,	Z = -244.833  mm,
	W = 0.000 deg,	P = 30.000 deg,	R = 138.421 deg
};
P[117]{
   GP1:
	UF : 0, UT : 1,		CONFIG : 'N U T, 0, 0, 0',
	X = 1128.438  mm,	Y = -184.017  mm,	Z = -245.291  mm,
	W = 0.000 deg,	P = 30.000 deg,	R = 138.421 deg
};
P[118]{
   GP1:
	UF : 0, UT : 1,		CONFIG : 'N U T, 0, 0, 0',
	X = 1134.675  mm,	Y = -186.054  mm,	Z = -245.793  mm,
	W = 0.000 deg,	P = 30.000 deg,	R = 138.421 deg
};
P[119]{
   GP1:
	UF : 0, UT : 1,		CONFIG : 'N U T, 0, 0, 0',
	X = 1136.583  mm,	Y = -184.107  mm,	Z = -246.362  mm,
	W = 0.000 deg,	P = 30.000 deg,	R = 138.421 deg
};
P[120]{
   GP1:
	UF : 0, UT : 1,		CONFIG : 'N U T, 0, 0, 0',
	X = 1138.558  mm,	Y = -182.119  mm,	Z = -246.979  mm,
	W = 0.000 deg,	P = 30.000 deg,	R = 138.421 deg
};
P[121]{
   GP1:
	UF : 0, UT : 1,		CONFIG : 'N U T, 0, 0, 0',
	X = 1140.539  mm,	Y = -180.143  mm,	Z = -247.626  mm,
	W = 0.000 deg,	P = 30.000 deg,	R = 138.421 deg
};
P[122]{
   GP1:
	UF : 0, UT : 1,		CONFIG : 'N U T, 0, 0, 0',
	X = 1142.590  mm,	Y = -178.170  mm,	Z = -248.284  mm,
	W = 0.000 deg,	P = 30.000 deg,	R = 138.421 deg
};
P[123]{
   GP1:
	UF : 0, UT : 1,		CONFIG : 'N U T, 0, 0, 0',
	X = 1144.710  mm,	Y = -176.160  mm,	Z = -248.937  mm,
	W = 0.000 deg,	P = 30.000 deg,	R = 138.421 deg
};
P[124]{
   GP1:
	UF : 0, UT : 1,		CONFIG : 'N U T, 0, 0, 0',
	X = 1146.769  mm,	Y = -174.143  mm,	Z = -249.544  mm,
	W = 0.000 deg,	P = 30.000 deg,	R = 143.878 deg
};
P[125]{
   GP1:
	UF : 0, UT : 1,		CONFIG : 'N U T, 0, 0, 0',
	X = 1148.836  mm,	Y = -172.116  mm,	Z = -250.142  mm,
	W = 0.000 deg,	P = 30.000 deg,	R = 155.199 deg
};
P[126]{
   GP1:
	UF : 0, UT : 1,		CONFIG : 'N U T, 0, 0, 0',
	X = 1150.808  mm,	Y = -170.084  mm,	Z = -250.710  mm,
	W = 0.000 deg,	P = 30.000 deg,	R = 166.229 deg
};
P[127]{
   GP1:
	UF : 0, UT : 1,		CONFIG : 'N U T, 0, 0, 0',
	X = 1152.763  mm,	Y = -168.050  mm,	Z = -251.268  mm,
	W = 0.000 deg,	P = 30.000 deg,	R = 177.202 deg
};
P[128]{
   GP1:
	UF : 0, UT : 1,		CONFIG : 'N U T, 0, 0, 0',
	X = 1154.697  mm,	Y = -165.922  mm,	Z = -251.791  mm,
	W = 0.000 deg,	P = 30.000 deg,	R = 177.202 deg
};
P[129]{
   GP1:
	UF : 0, UT : 1,		CONFIG : 'N U T, 0, 0, 0',
	X = 1156.360  mm,	Y = -163.730  mm,	Z = -252.211  mm,
	W = 0.000 deg,	P = 30.000 deg,	R = 177.202 deg
};
P[130]{
   GP1:
	UF : 0, UT : 1,		CONFIG : 'N U T, 0, 0, 0',
	X = 1157.798  mm,	Y = -161.531  mm,	Z = -252.563  mm,
	W = 0.000 deg,	P = 30.000 deg,	R = 177.202 deg
};
P[131]{
   GP1:
	UF : 0, UT : 1,		CONFIG : 'N U T, 0, 0, 0',
	X = 1159.014  mm,	Y = -159.241  mm,	Z = -252.845  mm,
	W = 0.000 deg,	P = 30.000 deg,	R = 177.202 deg
};
P[132]{
   GP1:
	UF : 0, UT : 1,		CONFIG : 'N U T, 0, 0, 0',
	X = 1159.894  mm,	Y = -156.908  mm,	Z = -253.036  mm,
	W = 0.000 deg,	P = 30.000 deg,	R = 177.202 deg
};
P[133]{
   GP1:
	UF : 0, UT : 1,		CONFIG : 'N U T, 0, 0, 0',
	X = 1160.492  mm,	Y = -154.607  mm,	Z = -253.156  mm,
	W = 0.000 deg,	P = 30.000 deg,	R = 177.202 deg
};
P[134]{
   GP1:
	UF : 0, UT : 1,		CONFIG : 'N U T, 0, 0, 0',
	X = 1160.843  mm,	Y = -152.330  mm,	Z = -253.216  mm,
	W = 0.000 deg,	P = 30.000 deg,	R = 177.202 deg
};
P[135]{
   GP1:
	UF : 0, UT : 1,		CONFIG : 'N U T, 0, 0, 0',
	X = 1160.992  mm,	Y = -150.179  mm,	Z = -253.224  mm,
	W = 0.000 deg,	P = 30.000 deg,	R = 177.202 deg
};
P[136]{
   GP1:
	UF : 0, UT : 1,		CONFIG : 'N U T, 0, 0, 0',
	X = 1155.102  mm,	Y = -147.886  mm,	Z = -253.229  mm,
	W = 0.000 deg,	P = 30.000 deg,	R = 177.202 deg
};
P[137]{
   GP1:
	UF : 0, UT : 1,		CONFIG : 'N U T, 0, 0, 0',
	X = 1155.149  mm,	Y = -145.939  mm,	Z = -253.230  mm,
	W = 0.000 deg,	P = 30.000 deg,	R = 177.202 deg
};
P[138]{
   GP1:
	UF : 0, UT : 1,		CONFIG : 'N U T, 0, 0, 0',
	X = 1155.182  mm,	Y = -143.957  mm,	Z = -253.228  mm,
	W = 0.000 deg,	P = 30.000 deg,	R = 177.202 deg
};
P[139]{
   GP1:
	UF : 0, UT : 1,		CONFIG : 'N U T, 0, 0, 0',
	X = 1155.206  mm,	Y = -141.973  mm,	Z = -253.223  mm,
	W = 0.000 deg,	P = 30.000 deg,	R = 177.202 deg
};
P[140]{
   GP1:
	UF : 0, UT : 1,		CONFIG : 'N U T, 0, 0, 0',
	X = 1155.217  mm,	Y = -139.988  mm,	Z = -253.219  mm,
	W = 0.000 deg,	P = 30.000 deg,	R = 177.202 deg
};
P[141]{
   GP1:
	UF : 0, UT : 1,		CONFIG : 'N U T, 0, 0, 0',
	X = 1155.222  mm,	Y = -137.995  mm,	Z = -253.216  mm,
	W = 0.000 deg,	P = 30.000 deg,	R = 177.202 deg
};
P[142]{
   GP1:
	UF : 0, UT : 1,		CONFIG : 'N U T, 0, 0, 0',
	X = 1155.224  mm,	Y = -136.000  mm,	Z = -253.205  mm,
	W = 0.000 deg,	P = 30.000 deg,	R = 177.202 deg
};
P[143]{
   GP1:
	UF : 0, UT : 1,		CONFIG : 'N U T, 0, 0, 0',
	X = 1155.222  mm,	Y = -134.001  mm,	Z = -253.179  mm,
	W = 0.000 deg,	P = 30.000 deg,	R = 177.202 deg
};
P[144]{
   GP1:
	UF : 0, UT : 1,		CONFIG : 'N U T, 0, 0, 0',
	X = 1155.222  mm,	Y = -132.000  mm,	Z = -253.151  mm,
	W = 0.000 deg,	P = 30.000 deg,	R = 177.202 deg
};
P[145]{
   GP1:
	UF : 0, UT : 1,		CONFIG : 'N U T, 0, 0, 0',
	X = 1155.222  mm,	Y = -130.005  mm,	Z = -253.118  mm,
	W = 0.000 deg,	P = 30.000 deg,	R = 177.202 deg
};
P[146]{
   GP1:
	UF : 0, UT : 1,		CONFIG : 'N U T, 0, 0, 0',
	X = 1155.216  mm,	Y = -128.018  mm,	Z = -253.083  mm,
	W = 0.000 deg,	P = 30.000 deg,	R = 177.202 deg
};
P[147]{
   GP1:
	UF : 0, UT : 1,		CONFIG : 'N U T, 0, 0, 0',
	X = 1155.198  mm,	Y = -126.034  mm,	Z = -253.044  mm,
	W = 0.000 deg,	P = 30.000 deg,	R = 177.202 deg
};
P[148]{
   GP1:
	UF : 0, UT : 1,		CONFIG : 'N U T, 0, 0, 0',
	X = 1155.171  mm,	Y = -124.047  mm,	Z = -252.999  mm,
	W = 0.000 deg,	P = 30.000 deg,	R = 177.202 deg
};
P[149]{
   GP1:
	UF : 0, UT : 1,		CONFIG : 'N U T, 0, 0, 0',
	X = 1155.136  mm,	Y = -122.066  mm,	Z = -252.958  mm,
	W = 0.000 deg,	P = 30.000 deg,	R = 177.202 deg
};
P[150]{
   GP1:
	UF : 0, UT : 1,		CONFIG : 'N U T, 0, 0, 0',
	X = 1155.084  mm,	Y = -120.098  mm,	Z = -252.918  mm,
	W = 0.000 deg,	P = 30.000 deg,	R = 177.202 deg
};
P[151]{
   GP1:
	UF : 0, UT : 1,		CONFIG : 'N U T, 0, 0, 0',
	X = 1155.007  mm,	Y = -118.127  mm,	Z = -252.871  mm,
	W = 0.000 deg,	P = 30.000 deg,	R = 177.202 deg
};
P[152]{
   GP1:
	UF : 0, UT : 1,		CONFIG : 'N U T, 0, 0, 0',
	X = 1154.917  mm,	Y = -116.143  mm,	Z = -252.825  mm,
	W = 0.000 deg,	P = 30.000 deg,	R = 177.202 deg
};
P[153]{
   GP1:
	UF : 0, UT : 1,		CONFIG : 'N U T, 0, 0, 0',
	X = 1154.818  mm,	Y = -114.172  mm,	Z = -252.777  mm,
	W = 0.000 deg,	P = 30.000 deg,	R = 177.202 deg
};
P[154]{
   GP1:
	UF : 0, UT : 1,		CONFIG : 'N U T, 0, 0, 0',
	X = 1154.691  mm,	Y = -112.211  mm,	Z = -252.715  mm,
	W = 0.000 deg,	P = 30.000 deg,	R = 177.202 deg
};
P[155]{
   GP1:
	UF : 0, UT : 1,		CONFIG : 'N U T, 0, 0, 0',
	X = 1160.516  mm,	Y = -109.701  mm,	Z = -252.645  mm,
	W = 0.000 deg,	P = 30.000 deg,	R = -173.956 deg
};
P[156]{
   GP1:
	UF : 0, UT : 1,		CONFIG : 'N U T, 0, 0, 0',
	X = 1160.262  mm,	Y = -107.642  mm,	Z = -252.545  mm,
	W = 0.000 deg,	P = 30.000 deg,	R = -164.439 deg
};
P[157]{
   GP1:
	UF : 0, UT : 1,		CONFIG : 'N U T, 0, 0, 0',
	X = 1160.025  mm,	Y = -105.618  mm,	Z = -252.454  mm,
	W = 0.000 deg,	P = 30.000 deg,	R = -154.933 deg
};
P[158]{
   GP1:
	UF : 0, UT : 1,		CONFIG : 'N U T, 0, 0, 0',
	X = 1159.714  mm,	Y = -103.422  mm,	Z = -252.349  mm,
	W = 0.000 deg,	P = 30.000 deg,	R = -145.395 deg
};
P[159]{
   GP1:
	UF : 0, UT : 1,		CONFIG : 'N U T, 0, 0, 0',
	X = 1159.128  mm,	Y = -101.106  mm,	Z = -252.180  mm,
	W = 0.000 deg,	P = 30.000 deg,	R = -135.632 deg
};
P[160]{
   GP1:
	UF : 0, UT : 1,		CONFIG : 'N U T, 0, 0, 0',
	X = 1158.244  mm,	Y = -98.741  mm,	Z = -251.933  mm,
	W = 0.000 deg,	P = 30.000 deg,	R = -135.632 deg
};
P[161]{
   GP1:
	UF : 0, UT : 1,		CONFIG : 'N U T, 0, 0, 0',
	X = 1156.927  mm,	Y = -96.361  mm,	Z = -251.584  mm,
	W = 0.000 deg,	P = 30.000 deg,	R = -135.632 deg
};
P[162]{
   GP1:
	UF : 0, UT : 1,		CONFIG : 'N U T, 0, 0, 0',
	X = 1155.304  mm,	Y = -94.190  mm,	Z = -251.115  mm,
	W = 0.000 deg,	P = 30.000 deg,	R = -135.632 deg
};
P[163]{
   GP1:
	UF : 0, UT : 1,		CONFIG : 'N U T, 0, 0, 0',
	X = 1153.661  mm,	Y = -92.042  mm,	Z = -250.643  mm,
	W = 0.000 deg,	P = 30.000 deg,	R = -135.632 deg
};
P[164]{
   GP1:
	UF : 0, UT : 1,		CONFIG : 'N U T, 0, 0, 0',
	X = 1151.648  mm,	Y = -89.942  mm,	Z = -250.029  mm,
	W = 0.000 deg,	P = 30.000 deg,	R = -135.632 deg
};
P[165]{
   GP1:
	UF : 0, UT : 1,		CONFIG : 'N U T, 0, 0, 0',
	X = 1149.827  mm,	Y = -87.972  mm,	Z = -249.440  mm,
	W = 0.000 deg,	P = 30.000 deg,	R = -135.632 deg
};
P[166]{
   GP1:
	UF : 0, UT : 1,		CONFIG : 'N U T, 0, 0, 0',
	X = 1143.687  mm,	Y = -90.133  mm,	Z = -248.856  mm,
	W = 0.000 deg,	P = 30.000 deg,	R = -135.632 deg
};
P[167]{
   GP1:
	UF : 0, UT : 1,		CONFIG : 'N U T, 0, 0, 0',
	X = 1141.508  mm,	Y = -88.179  mm,	Z = -248.141  mm,
	W = 0.000 deg,	P = 30.000 deg,	R = -135.632 deg
};
P[168]{
   GP1:
	UF : 0, UT : 1,		CONFIG : 'N U T, 0, 0, 0',
	X = 1139.519  mm,	Y = -86.192  mm,	Z = -247.482  mm,
	W = 0.000 deg,	P = 30.000 deg,	R = -135.632 deg
};
P[169]{
   GP1:
	UF : 0, UT : 1,		CONFIG : 'N U T, 0, 0, 0',
	X = 1137.314  mm,	Y = -84.256  mm,	Z = -246.699  mm,
	W = 0.000 deg,	P = 30.000 deg,	R = -135.632 deg
};
P[170]{
   GP1:
	UF : 0, UT : 1,		CONFIG : 'N U T, 0, 0, 0',
	X = 1134.981  mm,	Y = -82.215  mm,	Z = -245.920  mm,
	W = 0.000 deg,	P = 30.000 deg,	R = -135.632 deg
};
P[171]{
   GP1:
	UF : 0, UT : 1,		CONFIG : 'N U T, 0, 0, 0',
	X = 1132.990  mm,	Y = -80.304  mm,	Z = -245.251  mm,
	W = 0.000 deg,	P = 30.000 deg,	R = -135.632 deg
};
P[172]{
   GP1:
	UF : 0, UT : 1,		CONFIG : 'N U T, 0, 0, 0',
	X = 1130.415  mm,	Y = -78.407  mm,	Z = -244.456  mm,
	W = 0.000 deg,	P = 30.000 deg,	R = -139.273 deg
};
P[173]{
   GP1:
	UF : 0, UT : 1,		CONFIG : 'N U T, 0, 0, 0',
	X = 1127.594  mm,	Y = -76.290  mm,	Z = -243.695  mm,
	W = 0.000 deg,	P = 30.000 deg,	R = -154.647 deg
};
P[174]{
   GP1:
	UF : 0, UT : 1,		CONFIG : 'N U T, 0, 0, 0',
	X = 1125.363  mm,	Y = -74.125  mm,	Z = -243.137  mm,
	W = 0.000 deg,	P = 30.000 deg,	R = -167.752 deg
};
P[175]{
   GP1:
	UF : 0, UT : 1,		CONFIG : 'N U T, 0, 0, 0',
	X = 1123.193  mm,	Y = -71.896  mm,	Z = -242.638  mm,
	W = 0.000 deg,	P = 30.000 deg,	R = 179.467 deg
};
P[176]{
   GP1:
	UF : 0, UT : 1,		CONFIG : 'N U T, 0, 0, 0',
	X = 1121.669  mm,	Y = -69.579  mm,	Z = -242.391  mm,
	W = 0.000 deg,	P = 30.000 deg,	R = 179.467 deg
};
P[177]{
   GP1:
	UF : 0, UT : 1,		CONFIG : 'N U T, 0, 0, 0',
	X = 1120.401  mm,	Y = -67.423  mm,	Z = -242.178  mm,
	W = 0.000 deg,	P = 30.000 deg,	R = 179.467 deg
};
P[178]{
   GP1:
	UF : 0, UT : 1,		CONFIG : 'N U T, 0, 0, 0',
	X = 1119.222  mm,	Y = -64.956  mm,	Z = -241.992  mm,
	W = 0.000 deg,	P = 30.000 deg,	R = 179.467 deg
};
P[179]{
   GP1:
	UF : 0, UT : 1,		CONFIG : 'N U T, 0, 0, 0',
	X = 1118.727  mm,	Y = -62.420  mm,	Z = -241.930  mm,
	W = 0.000 deg,	P = 30.000 deg,	R = 179.467 deg
};
P[180]{
   GP1:
	UF : 0, UT : 1,		CONFIG : 'N U T, 0, 0, 0',
	X = 1118.512  mm,	Y = -60.268  mm,	Z = -241.899  mm,
	W = 0.000 deg,	P = 30.000 deg,	R = 179.467 deg
};
P[181]{
   GP1:
	UF : 0, UT : 1,		CONFIG : 'N U T, 0, 0, 0',
	X = 1118.344  mm,	Y = -58.174  mm,	Z = -241.879  mm,
	W = 0.000 deg,	P = 30.000 deg,	R = 179.467 deg
};
P[182]{
   GP1:
	UF : 0, UT : 1,		CONFIG : 'N U T, 0, 0, 0',
	X = 1118.269  mm,	Y = -56.077  mm,	Z = -241.866  mm,
	W = 0.000 deg,	P = 30.000 deg,	R = 179.467 deg
};
P[183]{
   GP1:
	UF : 0, UT : 1,		CONFIG : 'N U T, 0, 0, 0',
	X = 1118.236  mm,	Y = -54.036  mm,	Z = -241.854  mm,
	W = 0.000 deg,	P = 30.000 deg,	R = 179.467 deg
};
P[184]{
   GP1:
	UF : 0, UT : 1,		CONFIG : 'N U T, 0, 0, 0',
	X = 1118.219  mm,	Y = -52.018  mm,	Z = -241.835  mm,
	W = 0.000 deg,	P = 30.000 deg,	R = 179.467 deg
};
P[185]{
   GP1:
	UF : 0, UT : 1,		CONFIG : 'N U T, 0, 0, 0',
	X = 1118.211  mm,	Y = -50.009  mm,	Z = -241.819  mm,
	W = 0.000 deg,	P = 30.000 deg,	R = 179.467 deg
};
P[186]{
   GP1:
	UF : 0, UT : 1,		CONFIG : 'N U T, 0, 0, 0',
	X = 1118.207  mm,	Y = -48.002  mm,	Z = -241.807  mm,
	W = 0.000 deg,	P = 30.000 deg,	R = 179.467 deg
};
P[187]{
   GP1:
	UF : 0, UT : 1,		CONFIG : 'N U T, 0, 0, 0',
	X = 1118.208  mm,	Y = -45.995  mm,	Z = -241.800  mm,
	W = 0.000 deg,	P = 30.000 deg,	R = 179.467 deg
};
P[188]{
   GP1:
	UF : 0, UT : 1,		CONFIG : 'N U T, 0, 0, 0',
	X = 1118.214  mm,	Y = -43.990  mm,	Z = -241.797  mm,
	W = 0.000 deg,	P = 30.000 deg,	R = 179.467 deg
};
P[189]{
   GP1:
	UF : 0, UT : 1,		CONFIG : 'N U T, 0, 0, 0',
	X = 1118.222  mm,	Y = -41.987  mm,	Z = -241.786  mm,
	W = 0.000 deg,	P = 30.000 deg,	R = 179.467 deg
};
P[190]{
   GP1:
	UF : 0, UT : 1,		CONFIG : 'N U T, 0, 0, 0',
	X = 1118.231  mm,	Y = -39.984  mm,	Z = -241.774  mm,
	W = 0.000 deg,	P = 30.000 deg,	R = 179.467 deg
};
P[191]{
   GP1:
	UF : 0, UT : 1,		CONFIG : 'N U T, 0, 0, 0',
	X = 1118.243  mm,	Y = -37.974  mm,	Z = -241.771  mm,
	W = 0.000 deg,	P = 30.000 deg,	R = 179.467 deg
};
P[192]{
   GP1:
	UF : 0, UT : 1,		CONFIG : 'N U T, 0, 0, 0',
	X = 1124.265  mm,	Y = -36.040  mm,	Z = -241.762  mm,
	W = 0.000 deg,	P = 30.000 deg,	R = 179.467 deg
};
P[193]{
   GP1:
	UF : 0, UT : 1,		CONFIG : 'N U T, 0, 0, 0',
	X = 1124.296  mm,	Y = -34.057  mm,	Z = -241.754  mm,
	W = 0.000 deg,	P = 30.000 deg,	R = 179.467 deg
};
P[194]{
   GP1:
	UF : 0, UT : 1,		CONFIG : 'N U T, 0, 0, 0',
	X = 1124.340  mm,	Y = -32.077  mm,	Z = -241.742  mm,
	W = 0.000 deg,	P = 30.000 deg,	R = 179.467 deg
};
P[195]{
   GP1:
	UF : 0, UT : 1,		CONFIG : 'N U T, 0, 0, 0',
	X = 1124.397  mm,	Y = -30.097  mm,	Z = -241.715  mm,
	W = 0.000 deg,	P = 30.000 deg,	R = 179.467 deg
};
P[196]{
   GP1:
	UF : 0, UT : 1,		CONFIG : 'N U T, 0, 0, 0',
	X = 1124.468  mm,	Y = -28.109  mm,	Z = -241.696  mm,
	W = 0.000 deg,	P = 30.000 deg,	R = 179.467 deg
};
P[197]{
   GP1:
	UF : 0, UT : 1,		CONFIG : 'N U T, 0, 0, 0',
	X = 1124.541  mm,	Y = -26.126  mm,	Z = -241.679  mm,
	W = 0.000 deg,	P = 30.000 deg,	R = 179.467 deg
};
P[198]{
   GP1:
	UF : 0, UT : 1,		CONFIG : 'N U T, 0, 0, 0',
	X = 1124.634  mm,	Y = -24.145  mm,	Z = -241.661  mm,
	W = 0.000 deg,	P = 30.000 deg,	R = 179.467 deg
};
P[199]{
   GP1:
	UF : 0, UT : 1,		CONFIG : 'N U T, 0, 0, 0',
	X = 1124.733  mm,	Y = -22.171  mm,	Z = -241.647  mm,
	W = 0.000 deg,	P = 30.000 deg,	R = 179.467 deg
};
P[200]{
   GP1:
	UF : 0, UT : 1,		CONFIG : 'N U T, 0, 0, 0',
	X = 1124.859  mm,	Y = -20.212  mm,	Z = -241.628  mm,
	W = 0.000 deg,	P = 30.000 deg,	R = 179.467 deg
};
P[201]{
   GP1:
	UF : 0, UT : 1,		CONFIG : 'N U T, 0, 0, 0',
	X = 1125.010  mm,	Y = -18.254  mm,	Z = -241.612  mm,
	W = 0.000 deg,	P = 30.000 deg,	R = 179.467 deg
};
P[202]{
   GP1:
	UF : 0, UT : 1,		CONFIG : 'N U T, 0, 0, 0',
	X = 1119.229  mm,	Y = -15.638  mm,	Z = -241.608  mm,
	W = 0.000 deg,	P = 30.000 deg,	R = 171.877 deg
};
P[203]{
   GP1:
	UF : 0, UT : 1,		CONFIG : 'N U T, 0, 0, 0',
	X = 1119.551  mm,	Y = -13.487  mm,	Z = -241.620  mm,
	W = 0.000 deg,	P = 30.000 deg,	R = 163.298 deg
};
P[204]{
   GP1:
	UF : 0, UT : 1,		CONFIG : 'N U T, 0, 0, 0',
	X = 1119.969  mm,	Y = -11.364  mm,	Z = -241.648  mm,
	W = 0.000 deg,	P = 30.000 deg,	R = 154.650 deg
};
P[205]{
   GP1:
	UF : 0, UT : 1,		CONFIG : 'N U T, 0, 0, 0',
	X = 1120.480  mm,	Y = -9.211  mm,	Z = -241.691  mm,
	W = 0.000 deg,	P = 30.000 deg,	R = 145.928 deg
};
P[206]{
   GP1:
	UF : 0, UT : 1,		CONFIG : 'N U T, 0, 0, 0',
	X = 1121.164  mm,	Y = -6.995  mm,	Z = -241.766  mm,
	W = 0.000 deg,	P = 30.000 deg,	R = 137.045 deg
};
P[207]{
   GP1:
	UF : 0, UT : 1,		CONFIG : 'N U T, 0, 0, 0',
	X = 1122.079  mm,	Y = -4.729  mm,	Z = -241.911  mm,
	W = 0.000 deg,	P = 30.000 deg,	R = 137.045 deg
};
P[208]{
   GP1:
	UF : 0, UT : 1,		CONFIG : 'N U T, 0, 0, 0',
	X = 1123.258  mm,	Y = -2.508  mm,	Z = -242.096  mm,
	W = 0.000 deg,	P = 30.000 deg,	R = 137.045 deg
};
P[209]{
   GP1:
	UF : 0, UT : 1,		CONFIG : 'N U T, 0, 0, 0',
	X = 1124.574  mm,	Y = -0.365  mm,	Z = -242.323  mm,
	W = 0.000 deg,	P = 30.000 deg,	R = 137.045 deg
};
P[210]{
   GP1:
	UF : 0, UT : 1,		CONFIG : 'N U T, 0, 0, 0',
	X = 1126.076  mm,	Y = 1.819  mm,	Z = -242.609  mm,
	W = 0.000 deg,	P = 30.000 deg,	R = 137.045 deg
};
P[211]{
   GP1:
	UF : 0, UT : 1,		CONFIG : 'N U T, 0, 0, 0',
	X = 1127.885  mm,	Y = 3.980  mm,	Z = -243.015  mm,
	W = 0.000 deg,	P = 30.000 deg,	R = 137.045 deg
};
P[212]{
   GP1:
	UF : 0, UT : 1,		CONFIG : 'N U T, 0, 0, 0',
	X = 1134.158  mm,	Y = 1.942  mm,	Z = -243.499  mm,
	W = 0.000 deg,	P = 30.000 deg,	R = 137.045 deg
};
P[213]{
   GP1:
	UF : 0, UT : 1,		CONFIG : 'N U T, 0, 0, 0',
	X = 1136.052  mm,	Y = 3.900  mm,	Z = -244.042  mm,
	W = 0.000 deg,	P = 30.000 deg,	R = 137.045 deg
};
P[214]{
   GP1:
	UF : 0, UT : 1,		CONFIG : 'N U T, 0, 0, 0',
	X = 1138.003  mm,	Y = 5.863  mm,	Z = -244.600  mm,
	W = 0.000 deg,	P = 30.000 deg,	R = 137.045 deg
};
P[215]{
   GP1:
	UF : 0, UT : 1,		CONFIG : 'N U T, 0, 0, 0',
	X = 1140.023  mm,	Y = 7.812  mm,	Z = -245.234  mm,
	W = 0.000 deg,	P = 30.000 deg,	R = 137.045 deg
};
P[216]{
   GP1:
	UF : 0, UT : 1,		CONFIG : 'N U T, 0, 0, 0',
	X = 1142.195  mm,	Y = 9.793  mm,	Z = -245.934  mm,
	W = 0.000 deg,	P = 30.000 deg,	R = 137.045 deg
};
P[217]{
   GP1:
	UF : 0, UT : 1,		CONFIG : 'N U T, 0, 0, 0',
	X = 1144.380  mm,	Y = 11.825  mm,	Z = -246.632  mm,
	W = 0.000 deg,	P = 30.000 deg,	R = 137.045 deg
};
P[218]{
   GP1:
	UF : 0, UT : 1,		CONFIG : 'N U T, 0, 0, 0',
	X = 1146.443  mm,	Y = 13.830  mm,	Z = -247.285  mm,
	W = 0.000 deg,	P = 30.000 deg,	R = 140.932 deg
};
P[219]{
   GP1:
	UF : 0, UT : 1,		CONFIG : 'N U T, 0, 0, 0',
	X = 1148.536  mm,	Y = 15.794  mm,	Z = -247.940  mm,
	W = 0.000 deg,	P = 30.000 deg,	R = 152.770 deg
};
P[220]{
   GP1:
	UF : 0, UT : 1,		CONFIG : 'N U T, 0, 0, 0',
	X = 1150.754  mm,	Y = 17.802  mm,	Z = -248.610  mm,
	W = 0.000 deg,	P = 30.000 deg,	R = 164.844 deg
};
P[221]{
   GP1:
	UF : 0, UT : 1,		CONFIG : 'N U T, 0, 0, 0',
	X = 1152.927  mm,	Y = 19.875  mm,	Z = -249.243  mm,
	W = 0.000 deg,	P = 30.000 deg,	R = 176.569 deg
};
P[222]{
   GP1:
	UF : 0, UT : 1,		CONFIG : 'N U T, 0, 0, 0',
	X = 1154.952  mm,	Y = 21.987  mm,	Z = -249.811  mm,
	W = 0.000 deg,	P = 30.000 deg,	R = 176.569 deg
};
P[223]{
   GP1:
	UF : 0, UT : 1,		CONFIG : 'N U T, 0, 0, 0',
	X = 1156.766  mm,	Y = 24.116  mm,	Z = -250.305  mm,
	W = 0.000 deg,	P = 30.000 deg,	R = 176.569 deg
};
P[224]{
   GP1:
	UF : 0, UT : 1,		CONFIG : 'N U T, 0, 0, 0',
	X = 1158.424  mm,	Y = 26.293  mm,	Z = -250.738  mm,
	W = 0.000 deg,	P = 30.000 deg,	R = 176.569 deg
};
P[225]{
   GP1:
	UF : 0, UT : 1,		CONFIG : 'N U T, 0, 0, 0',
	X = 1159.841  mm,	Y = 28.580  mm,	Z = -251.084  mm,
	W = 0.000 deg,	P = 30.000 deg,	R = 176.569 deg
};
P[226]{
   GP1:
	UF : 0, UT : 1,		CONFIG : 'N U T, 0, 0, 0',
	X = 1160.920  mm,	Y = 30.959  mm,	Z = -251.337  mm,
	W = 0.000 deg,	P = 30.000 deg,	R = 176.569 deg
};
P[227]{
   GP1:
	UF : 0, UT : 1,		CONFIG : 'N U T, 0, 0, 0',
	X = 1161.593  mm,	Y = 33.286  mm,	Z = -251.491  mm,
	W = 0.000 deg,	P = 30.000 deg,	R = 176.569 deg
};
P[228]{
   GP1:
	UF : 0, UT : 1,		CONFIG : 'N U T, 0, 0, 0',
	X = 1162.051  mm,	Y = 35.542  mm,	Z = -251.603  mm,
	W = 0.000 deg,	P = 30.000 deg,	R = 176.569 deg
};
P[229]{
   GP1:
	UF : 0, UT : 1,		CONFIG : 'N U T, 0, 0, 0',
	X = 1162.287  mm,	Y = 37.766  mm,	Z = -251.657  mm,
	W = 0.000 deg,	P = 30.000 deg,	R = 176.569 deg
};
P[230]{
   GP1:
	UF : 0, UT : 1,		CONFIG : 'N U T, 0, 0, 0',
	X = 1156.401  mm,	Y = 40.114  mm,	Z = -251.674  mm,
	W = 0.000 deg,	P = 30.000 deg,	R = 176.569 deg
};
P[231]{
   GP1:
	UF : 0, UT : 1,		CONFIG : 'N U T, 0, 0, 0',
	X = 1156.449  mm,	Y = 42.058  mm,	Z = -251.677  mm,
	W = 0.000 deg,	P = 30.000 deg,	R = 176.569 deg
};
P[232]{
   GP1:
	UF : 0, UT : 1,		CONFIG : 'N U T, 0, 0, 0',
	X = 1156.477  mm,	Y = 44.039  mm,	Z = -251.670  mm,
	W = 0.000 deg,	P = 30.000 deg,	R = 176.569 deg
};
P[233]{
   GP1:
	UF : 0, UT : 1,		CONFIG : 'N U T, 0, 0, 0',
	X = 1156.501  mm,	Y = 46.037  mm,	Z = -251.660  mm,
	W = 0.000 deg,	P = 30.000 deg,	R = 176.569 deg
};
P[234]{
   GP1:
	UF : 0, UT : 1,		CONFIG : 'N U T, 0, 0, 0',
	X = 1156.526  mm,	Y = 48.032  mm,	Z = -251.643  mm,
	W = 0.000 deg,	P = 30.000 deg,	R = 176.569 deg
};
P[235]{
   GP1:
	UF : 0, UT : 1,		CONFIG : 'N U T, 0, 0, 0',
	X = 1156.544  mm,	Y = 50.024  mm,	Z = -251.621  mm,
	W = 0.000 deg,	P = 30.000 deg,	R = 176.569 deg
};
P[236]{
   GP1:
	UF : 0, UT : 1,		CONFIG : 'N U T, 0, 0, 0',
	X = 1156.558  mm,	Y = 52.013  mm,	Z = -251.597  mm,
	W = 0.000 deg,	P = 30.000 deg,	R = 176.569 deg
};
P[237]{
   GP1:
	UF : 0, UT : 1,		CONFIG : 'N U T, 0, 0, 0',
	X = 1156.561  mm,	Y = 54.001  mm,	Z = -251.570  mm,
	W = 0.000 deg,	P = 30.000 deg,	R = 176.569 deg
};
P[238]{
   GP1:
	UF : 0, UT : 1,		CONFIG : 'N U T, 0, 0, 0',
	X = 1156.559  mm,	Y = 55.993  mm,	Z = -251.544  mm,
	W = 0.000 deg,	P = 30.000 deg,	R = 176.569 deg
};
P[239]{
   GP1:
	UF : 0, UT : 1,		CONFIG : 'N U T, 0, 0, 0',
	X = 1156.552  mm,	Y = 57.985  mm,	Z = -251.519  mm,
	W = 0.000 deg,	P = 30.000 deg,	R = 176.569 deg
};
P[240]{
   GP1:
	UF : 0, UT : 1,		CONFIG : 'N U T, 0, 0, 0',
	X = 1156.539  mm,	Y = 59.978  mm,	Z = -251.490  mm,
	W = 0.000 deg,	P = 30.000 deg,	R = 176.569 deg
};
P[241]{
   GP1:
	UF : 0, UT : 1,		CONFIG : 'N U T, 0, 0, 0',
	X = 1156.523  mm,	Y = 61.970  mm,	Z = -251.462  mm,
	W = 0.000 deg,	P = 30.000 deg,	R = 176.569 deg
};
P[242]{
   GP1:
	UF : 0, UT : 1,		CONFIG : 'N U T, 0, 0, 0',
	X = 1156.499  mm,	Y = 63.957  mm,	Z = -251.429  mm,
	W = 0.000 deg,	P = 30.000 deg,	R = 176.569 deg
};
P[243]{
   GP1:
	UF : 0, UT : 1,		CONFIG : 'N U T, 0, 0, 0',
	X = 1156.466  mm,	Y = 65.941  mm,	Z = -251.392  mm,
	W = 0.000 deg,	P = 30.000 deg,	R = 176.569 deg
};
P[244]{
   GP1:
	UF : 0, UT : 1,		CONFIG : 'N U T, 0, 0, 0',
	X = 1156.422  mm,	Y = 67.924  mm,	Z = -251.358  mm,
	W = 0.000 deg,	P = 30.000 deg,	R = 176.569 deg
};
P[245]{
   GP1:
	UF : 0, UT : 1,		CONFIG : 'N U T, 0, 0, 0',
	X = 1156.365  mm,	Y = 69.911  mm,	Z = -251.317  mm,
	W = 0.000 deg,	P = 30.000 deg,	R = 176.569 deg
};
P[246]{
   GP1:
	UF : 0, UT : 1,		CONFIG : 'N U T, 0, 0, 0',
	X = 1156.304  mm,	Y = 71.904  mm,	Z = -251.276  mm,
	W = 0.000 deg,	P = 30.000 deg,	R = 176.569 deg
};
P[247]{
   GP1:
	UF : 0, UT : 1,		CONFIG : 'N U T, 0, 0, 0',
	X = 1156.237  mm,	Y = 73.889  mm,	Z = -251.236  mm,
	W = 0.000 deg,	P = 30.000 deg,	R = 176.569 deg
};
P[248]{
   GP1:
	UF : 0, UT : 1,		CONFIG : 'N U T, 0, 0, 0',
	X = 1156.157  mm,	Y = 75.874  mm,	Z = -251.194  mm,
	W = 0.000 deg,	P = 30.000 deg,	R = 176.569 deg
};
P[249]{
   GP1:
	UF : 0, UT : 1,		CONFIG : 'N U T, 0, 0, 0',
	X = 1156.069  mm,	Y = 77.865  mm,	Z = -251.146  mm,
	W = 0.000 deg,	P = 30.000 deg,	R = 176.569 deg
};
P[250]{
   GP1:
	UF : 0, UT : 1,		CONFIG : 'N U T, 0, 0, 0',
	X = 1161.969  mm,	Y = 80.180  mm,	Z = -251.103  mm,
	W = 0.000 deg,	P = 30.000 deg,	R = -174.990 deg
};
P[251]{
   GP1:
	UF : 0, UT : 1,		CONFIG : 'N U T, 0, 0, 0',
	X = 1161.809  mm,	Y = 82.304  mm,	Z = -251.035  mm,
	W = 0.000 deg,	P = 30.000 deg,	R = -165.533 deg
};
P[252]{
   GP1:
	UF : 0, UT : 1,		CONFIG : 'N U T, 0, 0, 0',
	X = 1161.525  mm,	Y = 84.502  mm,	Z = -250.942  mm,
	W = 0.000 deg,	P = 30.000 deg,	R = -156.020 deg
};
P[253]{
   GP1:
	UF : 0, UT : 1,		CONFIG : 'N U T, 0, 0, 0',
	X = 1161.033  mm,	Y = 86.815  mm,	Z = -250.798  mm,
	W = 0.000 deg,	P = 30.000 deg,	R = -146.363 deg
};
P[254]{
   GP1:
	UF : 0, UT : 1,		CONFIG : 'N U T, 0, 0, 0',
	X = 1160.256  mm,	Y = 89.029  mm,	Z = -250.564  mm,
	W = 0.000 deg,	P = 30.000 deg,	R = -136.305 deg
};
P[255]{
   GP1:
	UF : 0, UT : 1,		CONFIG : 'N U T, 0, 0, 0',
	X = 1159.401  mm,	Y = 91.274  mm,	Z = -250.315  mm,
	W = 0.000 deg,	P = 30.000 deg,	R = -136.305 deg
};
P[256]{
   GP1:
	UF : 0, UT : 1,		CONFIG : 'N U T, 0, 0, 0',
	X = 1158.064  mm,	Y = 93.656  mm,	Z = -249.956  mm,
	W = 0.000 deg,	P = 30.000 deg,	R = -136.305 deg
};
P[257]{
   GP1:
	UF : 0, UT : 1,		CONFIG : 'N U T, 0, 0, 0',
	X = 1156.402  mm,	Y = 95.847  mm,	Z = -249.467  mm,
	W = 0.000 deg,	P = 30.000 deg,	R = -136.305 deg
};
P[258]{
   GP1:
	UF : 0, UT : 1,		CONFIG : 'N U T, 0, 0, 0',
	X = 1154.613  mm,	Y = 98.065  mm,	Z = -248.950  mm,
	W = 0.000 deg,	P = 30.000 deg,	R = -136.305 deg
};
P[259]{
   GP1:
	UF : 0, UT : 1,		CONFIG : 'N U T, 0, 0, 0',
	X = 1148.179  mm,	Y = 95.824  mm,	Z = -248.226  mm,
	W = 0.000 deg,	P = 30.000 deg,	R = -136.305 deg
};
P[260]{
   GP1:
	UF : 0, UT : 1,		CONFIG : 'N U T, 0, 0, 0',
	X = 1146.088  mm,	Y = 97.893  mm,	Z = -247.560  mm,
	W = 0.000 deg,	P = 30.000 deg,	R = -136.305 deg
};
P[261]{
   GP1:
	UF : 0, UT : 1,		CONFIG : 'N U T, 0, 0, 0',
	X = 1144.252  mm,	Y = 99.804  mm,	Z = -246.921  mm,
	W = 0.000 deg,	P = 30.000 deg,	R = -136.305 deg
};
P[262]{
   GP1:
	UF : 0, UT : 1,		CONFIG : 'N U T, 0, 0, 0',
	X = 1141.895  mm,	Y = 101.790  mm,	Z = -246.117  mm,
	W = 0.000 deg,	P = 30.000 deg,	R = -136.305 deg
};
P[263]{
   GP1:
	UF : 0, UT : 1,		CONFIG : 'N U T, 0, 0, 0',
	X = 1139.890  mm,	Y = 103.808  mm,	Z = -245.435  mm,
	W = 0.000 deg,	P = 30.000 deg,	R = -136.305 deg
};
P[264]{
   GP1:
	UF : 0, UT : 1,		CONFIG : 'N U T, 0, 0, 0',
	X = 1137.742  mm,	Y = 105.678  mm,	Z = -244.641  mm,
	W = 0.000 deg,	P = 30.000 deg,	R = -136.305 deg
};
P[265]{
   GP1:
	UF : 0, UT : 1,		CONFIG : 'N U T, 0, 0, 0',
	X = 1135.100  mm,	Y = 107.718  mm,	Z = -243.822  mm,
	W = 0.000 deg,	P = 30.000 deg,	R = -136.305 deg
};
P[266]{
   GP1:
	UF : 0, UT : 1,		CONFIG : 'N U T, 0, 0, 0',
	X = 1132.971  mm,	Y = 109.750  mm,	Z = -243.205  mm,
	W = 0.000 deg,	P = 30.000 deg,	R = -136.305 deg
};
P[267]{
   GP1:
	UF : 0, UT : 1,		CONFIG : 'N U T, 0, 0, 0',
	X = 1130.588  mm,	Y = 111.696  mm,	Z = -242.530  mm,
	W = 0.000 deg,	P = 30.000 deg,	R = -136.305 deg
};
P[268]{
   GP1:
	UF : 0, UT : 1,		CONFIG : 'N U T, 0, 0, 0',
	X = 1128.113  mm,	Y = 113.806  mm,	Z = -241.891  mm,
	W = 0.000 deg,	P = 30.000 deg,	R = -145.370 deg
};
P[269]{
   GP1:
	UF : 0, UT : 1,		CONFIG : 'N U T, 0, 0, 0',
	X = 1126.068  mm,	Y = 115.908  mm,	Z = -241.428  mm,
	W = 0.000 deg,	P = 30.000 deg,	R = -158.342 deg
};
P[270]{
   GP1:
	UF : 0, UT : 1,		CONFIG : 'N U T, 0, 0, 0',
	X = 1123.923  mm,	Y = 118.126  mm,	Z = -240.961  mm,
	W = 0.000 deg,	P = 30.000 deg,	R = -171.353 deg
};
P[271]{
   GP1:
	UF : 0, UT : 1,		CONFIG : 'N U T, 0, 0, 0',
	X = 1122.355  mm,	Y = 120.623  mm,	Z = -240.736  mm,
	W = 0.000 deg,	P = 30.000 deg,	R = 177.777 deg
};
P[272]{
   GP1:
	UF : 0, UT : 1,		CONFIG : 'N U T, 0, 0, 0',
	X = 1121.376  mm,	Y = 122.986  mm,	Z = -240.585  mm,
	W = 0.000 deg,	P = 30.000 deg,	R = 177.777 deg
};
P[273]{
   GP1:
	UF : 0, UT : 1,		CONFIG : 'N U T, 0, 0, 0',
	X = 1120.654  mm,	Y = 125.353  mm,	Z = -240.466  mm,
	W = 0.000 deg,	P = 30.000 deg,	R = 177.777 deg
};
P[274]{
   GP1:
	UF : 0, UT : 1,		CONFIG : 'N U T, 0, 0, 0',
	X = 1120.334  mm,	Y = 127.678  mm,	Z = -240.402  mm,
	W = 0.000 deg,	P = 30.000 deg,	R = 177.777 deg
};
P[275]{
   GP1:
	UF : 0, UT : 1,		CONFIG : 'N U T, 0, 0, 0',
	X = 1120.157  mm,	Y = 129.824  mm,	Z = -240.357  mm,
	W = 0.000 deg,	P = 30.000 deg,	R = 177.777 deg
};
P[276]{
   GP1:
	UF : 0, UT : 1,		CONFIG : 'N U T, 0, 0, 0',
	X = 1120.083  mm,	Y = 131.901  mm,	Z = -240.319  mm,
	W = 0.000 deg,	P = 30.000 deg,	R = 177.777 deg
};
P[277]{
   GP1:
	UF : 0, UT : 1,		CONFIG : 'N U T, 0, 0, 0',
	X = 1120.021  mm,	Y = 133.922  mm,	Z = -240.270  mm,
	W = 0.000 deg,	P = 30.000 deg,	R = 177.777 deg
};
P[278]{
   GP1:
	UF : 0, UT : 1,		CONFIG : 'N U T, 0, 0, 0',
	X = 1119.978  mm,	Y = 135.952  mm,	Z = -240.219  mm,
	W = 0.000 deg,	P = 30.000 deg,	R = 177.777 deg
};
P[279]{
   GP1:
	UF : 0, UT : 1,		CONFIG : 'N U T, 0, 0, 0',
	X = 1119.956  mm,	Y = 137.973  mm,	Z = -240.169  mm,
	W = 0.000 deg,	P = 30.000 deg,	R = 177.777 deg
};
P[280]{
   GP1:
	UF : 0, UT : 1,		CONFIG : 'N U T, 0, 0, 0',
	X = 1119.942  mm,	Y = 139.982  mm,	Z = -240.122  mm,
	W = 0.000 deg,	P = 30.000 deg,	R = 177.777 deg
};
P[281]{
   GP1:
	UF : 0, UT : 1,		CONFIG : 'N U T, 0, 0, 0',
	X = 1119.932  mm,	Y = 141.991  mm,	Z = -240.079  mm,
	W = 0.000 deg,	P = 30.000 deg,	R = 177.777 deg
};
P[282]{
   GP1:
	UF : 0, UT : 1,		CONFIG : 'N U T, 0, 0, 0',
	X = 1119.931  mm,	Y = 144.012  mm,	Z = -240.048  mm,
	W = 0.000 deg,	P = 30.000 deg,	R = 177.777 deg
};
P[283]{
   GP1:
	UF : 0, UT : 1,		CONFIG : 'N U T, 0, 0, 0',
	X = 1119.948  mm,	Y = 146.028  mm,	Z = -240.015  mm,
	W = 0.000 deg,	P = 30.000 deg,	R = 177.777 deg
};
P[284]{
   GP1:
	UF : 0, UT : 1,		CONFIG : 'N U T, 0, 0, 0',
	X = 1119.968  mm,	Y = 148.044  mm,	Z = -239.997  mm,
	W = 0.000 deg,	P = 30.000 deg,	R = 177.777 deg
};
P[285]{
   GP1:
	UF : 0, UT : 1,		CONFIG : 'N U T, 0, 0, 0',
	X = 1120.007  mm,	Y = 150.060  mm,	Z = -239.987  mm,
	W = 0.000 deg,	P = 30.000 deg,	R = 177.777 deg
};
P[286]{
   GP1:
	UF : 0, UT : 1,		CONFIG : 'N U T, 0, 0, 0',
	X = 1120.048  mm,	Y = 152.063  mm,	Z = -239.982  mm,
	W = 0.000 deg,	P = 30.000 deg,	R = 177.777 deg
};
P[287]{
   GP1:
	UF : 0, UT : 1,		CONFIG : 'N U T, 0, 0, 0',
	X = 1120.091  mm,	Y = 154.072  mm,	Z = -239.978  mm,
	W = 0.000 deg,	P = 30.000 deg,	R = 177.777 deg
};
P[288]{
   GP1:
	UF : 0, UT : 1,		CONFIG : 'N U T, 0, 0, 0',
	X = 1120.144  mm,	Y = 156.082  mm,	Z = -239.975  mm,
	W = 0.000 deg,	P = 30.000 deg,	R = 177.777 deg
};
P[289]{
   GP1:
	UF : 0, UT : 1,		CONFIG : 'N U T, 0, 0, 0',
	X = 1120.200  mm,	Y = 158.088  mm,	Z = -239.976  mm,
	W = 0.000 deg,	P = 30.000 deg,	R = 177.777 deg
};
P[290]{
   GP1:
	UF : 0, UT : 1,		CONFIG : 'N U T, 0, 0, 0',
	X = 1126.258  mm,	Y = 159.883  mm,	Z = -239.982  mm,
	W = 0.000 deg,	P = 30.000 deg,	R = 177.777 deg
};
P[291]{
   GP1:
	UF : 0, UT : 1,		CONFIG : 'N U T, 0, 0, 0',
	X = 1126.352  mm,	Y = 161.861  mm,	Z = -239.991  mm,
	W = 0.000 deg,	P = 30.000 deg,	R = 177.777 deg
};
P[292]{
   GP1:
	UF : 0, UT : 1,		CONFIG : 'N U T, 0, 0, 0',
	X = 1126.442  mm,	Y = 163.847  mm,	Z = -239.996  mm,
	W = 0.000 deg,	P = 30.000 deg,	R = 177.777 deg
};
P[293]{
   GP1:
	UF : 0, UT : 1,		CONFIG : 'N U T, 0, 0, 0',
	X = 1126.554  mm,	Y = 165.815  mm,	Z = -240.001  mm,
	W = 0.000 deg,	P = 30.000 deg,	R = 177.777 deg
};
P[294]{
   GP1:
	UF : 0, UT : 1,		CONFIG : 'N U T, 0, 0, 0',
	X = 1126.684  mm,	Y = 167.772  mm,	Z = -240.006  mm,
	W = 0.000 deg,	P = 30.000 deg,	R = 177.777 deg
};
P[295]{
   GP1:
	UF : 0, UT : 1,		CONFIG : 'N U T, 0, 0, 0',
	X = 1126.851  mm,	Y = 169.720  mm,	Z = -240.012  mm,
	W = 0.000 deg,	P = 30.000 deg,	R = 177.777 deg
};
P[296]{
   GP1:
	UF : 0, UT : 1,		CONFIG : 'N U T, 0, 0, 0',
	X = 1121.086  mm,	Y = 172.324  mm,	Z = -240.016  mm,
	W = 0.000 deg,	P = 30.000 deg,	R = 170.319 deg
};
P[297]{
   GP1:
	UF : 0, UT : 1,		CONFIG : 'N U T, 0, 0, 0',
	X = 1121.323  mm,	Y = 174.380  mm,	Z = -240.019  mm,
	W = 0.000 deg,	P = 30.000 deg,	R = 162.126 deg
};
P[298]{
   GP1:
	UF : 0, UT : 1,		CONFIG : 'N U T, 0, 0, 0',
	X = 1121.626  mm,	Y = 176.535  mm,	Z = -240.024  mm,
	W = 0.000 deg,	P = 30.000 deg,	R = 153.908 deg
};
P[299]{
   GP1:
	UF : 0, UT : 1,		CONFIG : 'N U T, 0, 0, 0',
	X = 1122.119  mm,	Y = 178.752  mm,	Z = -240.041  mm,
	W = 0.000 deg,	P = 30.000 deg,	R = 145.570 deg
};
P[300]{
   GP1:
	UF : 0, UT : 1,		CONFIG : 'N U T, 0, 0, 0',
	X = 1122.788  mm,	Y = 181.009  mm,	Z = -240.082  mm,
	W = 0.000 deg,	P = 30.000 deg,	R = 137.083 deg
};
P[301]{
   GP1:
	UF : 0, UT : 1,		CONFIG : 'N U T, 0, 0, 0',
	X = 1123.729  mm,	Y = 183.261  mm,	Z = -240.179  mm,
	W = 0.000 deg,	P = 30.000 deg,	R = 137.083 deg
};
P[302]{
   GP1:
	UF : 0, UT : 1,		CONFIG : 'N U T, 0, 0, 0',
	X = 1124.840  mm,	Y = 185.451  mm,	Z = -240.355  mm,
	W = 0.000 deg,	P = 30.000 deg,	R = 137.083 deg
};
P[303]{
   GP1:
	UF : 0, UT : 1,		CONFIG : 'N U T, 0, 0, 0',
	X = 1126.161  mm,	Y = 187.657  mm,	Z = -240.574  mm,
	W = 0.000 deg,	P = 30.000 deg,	R = 137.083 deg
};
P[304]{
   GP1:
	UF : 0, UT : 1,		CONFIG : 'N U T, 0, 0, 0',
	X = 1127.755  mm,	Y = 189.850  mm,	Z = -240.850  mm,
	W = 0.000 deg,	P = 30.000 deg,	R = 137.083 deg
};
P[305]{
   GP1:
	UF : 0, UT : 1,		CONFIG : 'N U T, 0, 0, 0',
	X = 1129.515  mm,	Y = 191.949  mm,	Z = -241.203  mm,
	W = 0.000 deg,	P = 30.000 deg,	R = 137.083 deg
};
P[306]{
   GP1:
	UF : 0, UT : 1,		CONFIG : 'N U T, 0, 0, 0',
	X = 1131.302  mm,	Y = 194.004  mm,	Z = -241.636  mm,
	W = 0.000 deg,	P = 30.000 deg,	R = 137.083 deg
};
P[307]{
   GP1:
	UF : 0, UT : 1,		CONFIG : 'N U T, 0, 0, 0',
	X = 1137.571  mm,	Y = 191.943  mm,	Z = -242.144  mm,
	W = 0.000 deg,	P = 30.000 deg,	R = 137.083 deg
};
P[308]{
   GP1:
	UF : 0, UT : 1,		CONFIG : 'N U T, 0, 0, 0',
	X = 1139.410  mm,	Y = 193.864  mm,	Z = -242.710  mm,
	W = 0.000 deg,	P = 30.000 deg,	R = 137.083 deg
};
P[309]{
   GP1:
	UF : 0, UT : 1,		CONFIG : 'N U T, 0, 0, 0',
	X = 1141.477  mm,	Y = 195.796  mm,	Z = -243.336  mm,
	W = 0.000 deg,	P = 30.000 deg,	R = 137.083 deg
};
P[310]{
   GP1:
	UF : 0, UT : 1,		CONFIG : 'N U T, 0, 0, 0',
	X = 1143.676  mm,	Y = 197.803  mm,	Z = -244.010  mm,
	W = 0.000 deg,	P = 30.000 deg,	R = 137.083 deg
};
P[311]{
   GP1:
	UF : 0, UT : 1,		CONFIG : 'N U T, 0, 0, 0',
	X = 1145.785  mm,	Y = 199.804  mm,	Z = -244.690  mm,
	W = 0.000 deg,	P = 30.000 deg,	R = 139.787 deg
};
P[312]{
   GP1:
	UF : 0, UT : 1,		CONFIG : 'N U T, 0, 0, 0',
	X = 1147.940  mm,	Y = 201.772  mm,	Z = -245.410  mm,
	W = 0.000 deg,	P = 30.000 deg,	R = 149.980 deg
};
P[313]{
   GP1:
	UF : 0, UT : 1,		CONFIG : 'N U T, 0, 0, 0',
	X = 1150.185  mm,	Y = 203.772  mm,	Z = -246.136  mm,
	W = 0.000 deg,	P = 30.000 deg,	R = 160.313 deg
};
P[314]{
   GP1:
	UF : 0, UT : 1,		CONFIG : 'N U T, 0, 0, 0',
	X = 1152.406  mm,	Y = 205.801  mm,	Z = -246.830  mm,
	W = 0.000 deg,	P = 30.000 deg,	R = 170.488 deg
};
P[315]{
   GP1:
	UF : 0, UT : 1,		CONFIG : 'N U T, 0, 0, 0',
	X = 1154.581  mm,	Y = 207.853  mm,	Z = -247.498  mm,
	W = 0.000 deg,	P = 30.000 deg,	R = 170.488 deg
};
P[316]{
   GP1:
	UF : 0, UT : 1,		CONFIG : 'N U T, 0, 0, 0',
	X = 1156.633  mm,	Y = 209.926  mm,	Z = -248.107  mm,
	W = 0.000 deg,	P = 30.000 deg,	R = 170.488 deg
};
P[317]{
   GP1:
	UF : 0, UT : 1,		CONFIG : 'N U T, 0, 0, 0',
	X = 1158.555  mm,	Y = 212.007  mm,	Z = -248.669  mm,
	W = 0.000 deg,	P = 30.000 deg,	R = 170.488 deg
};
P[318]{
   GP1:
	UF : 0, UT : 1,		CONFIG : 'N U T, 0, 0, 0',
	X = 1160.407  mm,	Y = 214.184  mm,	Z = -249.179  mm,
	W = 0.000 deg,	P = 30.000 deg,	R = 170.488 deg
};
P[319]{
   GP1:
	UF : 0, UT : 1,		CONFIG : 'N U T, 0, 0, 0',
	X = 1161.932  mm,	Y = 216.466  mm,	Z = -249.571  mm,
	W = 0.000 deg,	P = 30.000 deg,	R = 170.488 deg
};
P[320]{
   GP1:
	UF : 0, UT : 1,		CONFIG : 'N U T, 0, 0, 0',
	X = 1163.120  mm,	Y = 218.734  mm,	Z = -249.867  mm,
	W = 0.000 deg,	P = 30.000 deg,	R = 170.488 deg
};
P[321]{
   GP1:
	UF : 0, UT : 1,		CONFIG : 'N U T, 0, 0, 0',
	X = 1164.055  mm,	Y = 221.026  mm,	Z = -250.095  mm,
	W = 0.000 deg,	P = 30.000 deg,	R = 170.488 deg
};
P[322]{
   GP1:
	UF : 0, UT : 1,		CONFIG : 'N U T, 0, 0, 0',
	X = 1164.714  mm,	Y = 223.408  mm,	Z = -250.235  mm,
	W = 0.000 deg,	P = 30.000 deg,	R = 170.488 deg
};
P[323]{
   GP1:
	UF : 0, UT : 1,		CONFIG : 'N U T, 0, 0, 0',
	X = 1159.035  mm,	Y = 226.268  mm,	Z = -250.291  mm,
	W = 0.000 deg,	P = 30.000 deg,	R = 170.488 deg
};
P[324]{
   GP1:
	UF : 0, UT : 1,		CONFIG : 'N U T, 0, 0, 0',
	X = 1159.133  mm,	Y = 228.092  mm,	Z = -250.299  mm,
	W = 0.000 deg,	P = 30.000 deg,	R = 170.488 deg
};
P[325]{
   GP1:
	UF : 0, UT : 1,		CONFIG : 'N U T, 0, 0, 0',
	X = 1159.146  mm,	Y = 230.004  mm,	Z = -250.293  mm,
	W = 0.000 deg,	P = 30.000 deg,	R = 170.488 deg
};
P[326]{
   GP1:
	UF : 0, UT : 1,		CONFIG : 'N U T, 0, 0, 0',
	X = 1159.138  mm,	Y = 231.982  mm,	Z = -250.279  mm,
	W = 0.000 deg,	P = 30.000 deg,	R = 170.488 deg
};
P[327]{
   GP1:
	UF : 0, UT : 1,		CONFIG : 'N U T, 0, 0, 0',
	X = 1159.123  mm,	Y = 233.974  mm,	Z = -250.262  mm,
	W = 0.000 deg,	P = 30.000 deg,	R = 170.488 deg
};
P[328]{
   GP1:
	UF : 0, UT : 1,		CONFIG : 'N U T, 0, 0, 0',
	X = 1159.103  mm,	Y = 235.967  mm,	Z = -250.241  mm,
	W = 0.000 deg,	P = 30.000 deg,	R = 170.488 deg
};
P[329]{
   GP1:
	UF : 0, UT : 1,		CONFIG : 'N U T, 0, 0, 0',
	X = 1159.078  mm,	Y = 237.961  mm,	Z = -250.205  mm,
	W = 0.000 deg,	P = 30.000 deg,	R = 170.488 deg
};
P[330]{
   GP1:
	UF : 0, UT : 1,		CONFIG : 'N U T, 0, 0, 0',
	X = 1159.051  mm,	Y = 239.955  mm,	Z = -250.163  mm,
	W = 0.000 deg,	P = 30.000 deg,	R = 170.488 deg
};
P[331]{
   GP1:
	UF : 0, UT : 1,		CONFIG : 'N U T, 0, 0, 0',
	X = 1159.019  mm,	Y = 241.953  mm,	Z = -250.122  mm,
	W = 0.000 deg,	P = 30.000 deg,	R = 170.488 deg
};
P[332]{
   GP1:
	UF : 0, UT : 1,		CONFIG : 'N U T, 0, 0, 0',
	X = 1158.988  mm,	Y = 243.953  mm,	Z = -250.082  mm,
	W = 0.000 deg,	P = 30.000 deg,	R = 170.488 deg
};
P[333]{
   GP1:
	UF : 0, UT : 1,		CONFIG : 'N U T, 0, 0, 0',
	X = 1158.956  mm,	Y = 245.947  mm,	Z = -250.042  mm,
	W = 0.000 deg,	P = 30.000 deg,	R = 170.488 deg
};
P[334]{
   GP1:
	UF : 0, UT : 1,		CONFIG : 'N U T, 0, 0, 0',
	X = 1158.918  mm,	Y = 247.935  mm,	Z = -250.000  mm,
	W = 0.000 deg,	P = 30.000 deg,	R = 170.488 deg
};
P[335]{
   GP1:
	UF : 0, UT : 1,		CONFIG : 'N U T, 0, 0, 0',
	X = 1158.870  mm,	Y = 249.929  mm,	Z = -249.956  mm,
	W = 0.000 deg,	P = 30.000 deg,	R = 170.488 deg
};
P[336]{
   GP1:
	UF : 0, UT : 1,		CONFIG : 'N U T, 0, 0, 0',
	X = 1158.825  mm,	Y = 251.930  mm,	Z = -249.927  mm,
	W = 0.000 deg,	P = 30.000 deg,	R = 170.488 deg
};
P[337]{
   GP1:
	UF : 0, UT : 1,		CONFIG : 'N U T, 0, 0, 0',
	X = 1158.776  mm,	Y = 253.927  mm,	Z = -249.906  mm,
	W = 0.000 deg,	P = 30.000 deg,	R = 170.488 deg
};
/END
